Universal Robots URScript: Floor Straight.script

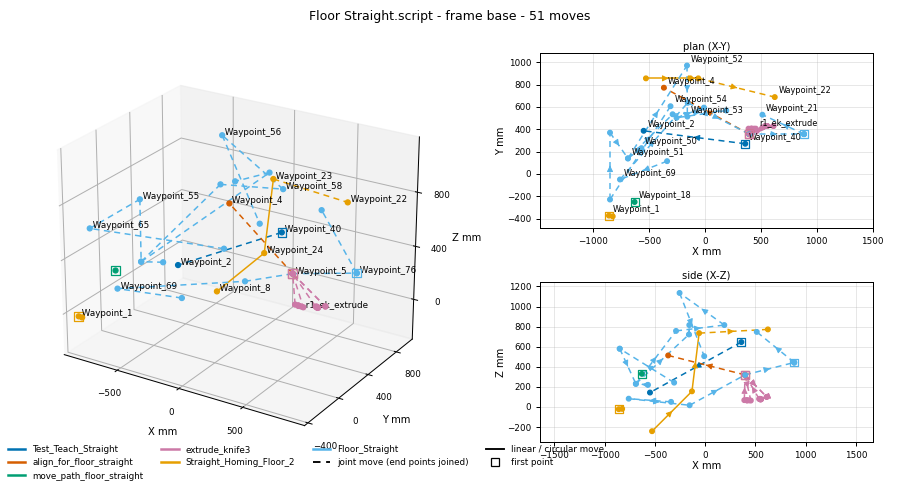
[picture p0: tool path of Floor Straight.script in frame base, 51 of 94 moves have a stored position in this frame; points joined in program order, loops and branches not executed]
def Floor_Straight():
  global _hidden_verificationVariable=0
  set_standard_analog_input_domain(0, 1)
  set_standard_analog_input_domain(1, 1)
  set_tool_analog_input_domain(0, 1)
  set_tool_analog_input_domain(1, 1)
  set_analog_outputdomain(0, 0)
  set_analog_outputdomain(1, 0)
  set_input_actions_to_default()
  set_target_payload(10.800000, [-0.001000, -0.053000, 0.068000], [0.081228, 0.081228, 0.081228, 0.000000, 0.000000, 0.000000])
  set_tool_communication(False, 115200, 0, 1, 1.5, 3.5)
  set_tool_output_mode(0)
  set_tool_digital_output_mode(0, 1)
  set_tool_digital_output_mode(1, 1)
  set_tool_voltage(0)
  set_tcp(p[-0.011699999999999999,-0.328,0.105,1.2092,-1.2092,1.2092])
  set_safety_mode_transition_hardness(1)
  set_gravity([0.0, 0.0, 9.82])
  global robot_number=3
  global Point_1=p[0.0,0.0,0.0,0.0,0.0,0.0]
  global Point_2=p[0.0,0.0,0.0,0.0,0.0,0.0]
  # begin: URCap Installation Node
  #   Source: UR Connect, 1.13.79, Universal Robots
  #   Type: UR Connect
  myurRPC = rpc_factory("xmlrpc","http://127.0.0.1:40474")
  # end: URCap Installation Node
  # begin: URCap Installation Node
  #   Source: MachineLogic for Universal Robots, 3.1.7, Vention Inc.
  #   Type: MachineLogic for Universal Robots
  def waitForResponse(expected_response_vention, cname_vention):
  response_vention = socket_read_string(cname_vention,timeout=15)
  while response_vention != expected_response_vention:
  sleep(0.01)
  response_vention = socket_read_string(cname_vention,timeout=15)
  end
  sleep(0.01)
  sync()
  end
  def sendString(string_vention, expected_response_vention, cname_vention):
  socket_send_string(str_cat(string_vention,";"), cname_vention)
  response_vention = socket_read_string(cname_vention,timeout=15)
  if(response_vention == "nAck"):
  popup("nAck received")
  end
  while response_vention != expected_response_vention:
  sleep(0.01)
  response_vention = socket_read_string(cname_vention,timeout=15)
  if(response_vention == "nAck"):
  popup("nAck received")
  end
  end
  sleep(0.01)
  sync()
  end
  def sendStringNAck(string_vention, expected_response_vention, cname_vention):
  socket_send_string(str_cat(string_vention,";"), cname_vention)
  response_vention = socket_read_string(cname_vention,timeout=15)
  if(response_vention == "nAck"):
  popup("nAck received")
  end
  while(response_vention != expected_response_vention and response_vention != "nAck"):
  sleep(0.01)
  response_vention = socket_read_string(cname_vention,timeout=15)
  if(response_vention == "nAck"):
  popup("nAck received",blocking=True)
  end
  end
  sleep(0.01)
  sync()
  end
  def sendStringWithTimeout(string_vention, expected_response_vention, cname_vention):
  socket_send_string(str_cat(string_vention,";"), cname_vention)
  response_vention = socket_read_string(cname_vention,timeout=10)
  if(response_vention == "nAck"):
  popup("nAck received"+string_vention)
  end
  sleep(0.01)
  sync()
  end
  def pollString(string_vention, expected_response_vention, cname_vention):
  socket_send_string(str_cat(string_vention,";"), cname_vention)
  response_vention = socket_read_string(cname_vention,timeout=15)
  if(response_vention == "nAck"):
  popup("nAck received")
  end
  while response_vention != expected_response_vention:
  sleep(1)
  socket_send_string(str_cat(string_vention,";"), cname_vention)
  response_vention = socket_read_string(cname_vention,timeout=15)
  if(response_vention == "nAck"):
  popup("nAck received")
  end
  end
  sleep(0.01)
  sync()
  end
  def sendVariable(var_vention, data_vention, expected_response_vention, cname_vention):
  socket_set_var(var_vention, data_vention, cname_vention)
  response_vention = socket_read_string(cname_vention,timeout=15)
  if(response_vention == "nAck"):
  popup("nAck received")
  end
  while response_vention != expected_response_vention:
  sleep(0.01)
  response_vention = socket_read_string(cname_vention,timeout=15)
  if(response_vention == "nAck"):
  popup("nAck received")
  end
  end
  sleep(0.01)
  sync()
  end
  def intToString(integer_vention,cname_vention):
  stringFix=""
  multiplier_vention123=1
  if integer_vention<0:
  stringFix="-"
  multiplier_vention123=-1
  end
  socket_set_var("GetString",integer_vention*multiplier_vention123,cname_vention)
  string_vention=""
  while string_vention=="":
  sleep(0.01)
  string_vention=socket_read_string(cname_vention,timeout=15)
  end
  sleep(0.01)
  sync()
  string_vention=stringFix+string_vention
  return string_vention
  end
  string_vention=""
  isVentionMovementBusy = False
  isVentionParallelMovementSendingScript = False
  ventionThreadHandle = 1
  isVentionMovementBusyMachineMotion1 = False
  isVentionParallelMovementSendingScriptMachineMotion1 = False
  socket_vention = socket_open("192.168.3.52", 9999, "MachineMotion1")
  if socket_vention==False:
  popup("Check configuration, can't connect to MachineMotion")
  end
  waitForResponse("MachineMotion connection established", "MachineMotion1")
  sendString("isReady", "MachineMotion isReady = true", "MachineMotion1")
  sendStringWithTimeout("setURCapVersion2", "setURCapVersion loaded", "MachineMotion1")
  sendString("SET speed_v2 1000000", "Ack", "MachineMotion1")
  sendString("SET acceleration_v2 100000", "Ack", "MachineMotion1")
  sendString("SET de_axis_1_microsteps_config 8", "Ack", "MachineMotion1")
  sendString("SET de_axis_1_mechanical_gain_config_v2 150000.0", "Ack", "MachineMotion1")
  sendString("SET de_axis_1_direction_config 1", "Ack", "MachineMotion1")
  sendString("SET de_axis_1_type_config Custom Actuator ", "Ack", "MachineMotion1")
  sendString("de_axis_1_config_exec", "Ack", "MachineMotion1")
  # end: URCap Installation Node
  # begin: URCap Installation Node
  #   Source: WireTank Serial, 4.9.0, WireTank, LLC
  #   Type: WireTank Serial
  WTSerialBridge = rpc_factory("xmlrpc","http://127.0.0.1:40511/RPC2")
  # end: URCap Installation Node
  step_count_93fcdbb1_1181_43ea_a7f0_580262fe9a13 = 0.0
  thread Step_Counter_Thread_773b6cc1_d8f8_46f9_9db1_b39c1ae6633a():
    while (True):
      step_count_93fcdbb1_1181_43ea_a7f0_580262fe9a13 = step_count_93fcdbb1_1181_43ea_a7f0_580262fe9a13 + 1.0
      sync()
    end
  end
  run Step_Counter_Thread_773b6cc1_d8f8_46f9_9db1_b39c1ae6633a()
  global free_dr_already=  False
  global freedrive_m_var=  False
  global Waypoint_76_p=p[.886939072471, .356263001241, .442999104957, 2.316306590719, 2.057646408592, .074101958719]
  global Waypoint_76_q=[-3.2647881984118814, -1.2522049299371645, 1.5824044773896437, 0.9175786249801816, -0.008369636028316307, -1.3112608249927966]
  global Waypoint_50_p=p[-.568711442653, .230601791901, .220208834751, -1.519093932087, -.535128035721, .573965472012]
  global Waypoint_50_q=[-0.021522347127095998, -1.2794721287539979, 2.4323821703540247, 5.090870934515753, -2.2996109167682093, 1.533644199371338]
  global Waypoint_51_p=p[-.689649894186, .139001107022, .230693120258, -.852023156701, -1.645963115617, 1.645984943001]
  global Waypoint_51_q=[-1.1454814116107386, -1.5427037247321387, 2.8454700152026575, 4.979047852545538, -4.902958456669943, 1.5718834400177002]
  global Waypoint_52_p=p[-.160992057407, .970528182050, .722037363514, -.554955923310, .106486629259, .328544950173]
  global Waypoint_52_q=[-1.2978580633746546, -1.3217003357461472, 2.2583277861224573, 3.7025129038044433, -2.952825371419088, 0.9627944231033325]
  global Waypoint_53_p=p[-.157624488365, .513351401913, .815670293526, -.672704566373, -1.852329693545, -.055423312366]
  global Waypoint_53_q=[-2.7676661650287073, -1.8206430874266566, 2.312763277684347, 1.0122546392628173, -1.0765226523028772, -0.8102834860431116]
  global Waypoint_54_p=p[-.308528116178, .606080777007, .242371251996, -2.133736658076, .349438277129, 2.130953356703]
  global Waypoint_54_q=[-1.9617512861834925, -1.2994225782207032, 2.207935158406393, 0.745708628291748, 1.5955500602722168, 1.41863214969635]
  global Waypoint_65_p=p[-.850299549699, -.229060500451, .580194265918, -.066683564301, -1.566406749139, -.045536147896]
  global Waypoint_65_q=[0.11527767777442932, -1.206728772526123, 2.660132948552267, 3.2525827127644042, -4.69939905801882, -0.18521625200380498]
  global Waypoint_55_p=p[-.850295942693, .369353811615, .580190947871, -.066690142153, -1.566409865149, -.045506050424]
  global Waypoint_55_q=[-0.89636737505068, -1.198587493305542, 2.6061368624316614, 3.3119169908710937, -4.700617257748739, 0.826545238494873]
  global Waypoint_59_p=p[-.689650832419, .138973473550, .230700469426, -.851985360280, -1.645991124348, 1.645990580233]
  global Waypoint_59_q=[-1.1454528013812464, -1.5427289356342335, 2.8454795519458216, 4.979044186859884, -4.902960960065023, 1.5718833208084106]
  global Waypoint_71_p=p[-.289684660393, .534258475721, .757199031184, -.295236718653, -.653013693815, .389426431276]
  global Waypoint_71_q=[-1.3941848913775843, -1.6550847492613734, 2.7336130777942103, 4.156678839320801, -3.798194471989767, 1.7310842275619507]
  global Waypoint_58_p=p[.191120239889, .567518478899, .815512910186, -.135765364935, .396070873472, .208834263225]
  global Waypoint_58_q=[-1.651280705128805, -1.7712346516051234, 2.617981735860006, 3.3066598612019042, -2.656208101903097, 0.8563313484191895]
  global Waypoint_56_p=p[-.254568281661, .502958752129, 1.135400507516, -.261908057482, -.749714619963, 1.349050618455]
  global Waypoint_56_q=[-2.0344861189471644, -1.9012485943236292, 2.469647232686178, 2.2012061315723876, -1.1677187124835413, -0.5094392935382288]
  global Waypoint_57_p=p[-.009221327687, .593713365169, .505808930157, -1.424394189587, -2.344106819810, -.527597949261]
  global Waypoint_57_q=[-2.920837704335348, -1.9932075939574183, 2.3856611887561243, 0.6815890508839111, -0.5688460508929651, -1.1506975332843226]
  global Waypoint_67_p=p[-.339169194335, .114271165560, .051007401747, -.434162127311, 1.872717119498, -1.885153895998]
  global Waypoint_67_q=[-1.410516087208883, -0.9778240484050293, 2.47756010690798, -1.72361483196401, -0.3956816832171839, 1.808600902557373]
  global Waypoint_69_p=p[-.760826542313, -.049762698068, .082649581767, -1.026233921905, -1.612699318499, 1.547123897415]
  global Waypoint_69_q=[-0.22154647508730108, -1.118469015961029, 2.7561236063586634, -1.5568565337783475, -3.851987902318136, 1.559481143951416]
  global Waypoint_70_p=p[-.154414768496, .636923137577, .016979120256, -.302753655748, 1.486961848367, .122240024639]
  global Waypoint_70_q=[-1.1281922499286097, -1.0678585332683106, 2.4290812651263636, -2.7994214497008265, -1.6034835020648401, 1.7401196956634521]
  global Waypoint_49_p=p[.397354147848, .356263001249, .319808682466, 2.316306590727, 2.057646408591, .074101958728]
  global Waypoint_49_q=[-3.4579480330096644, -2.0568953953185023, 2.3266006151782435, -0.2270372670939942, -0.1993797461139124, -0.10534602800478154]
  global Waypoint_75_p=p[.886939072471, .356263001241, .442999104957, 2.316306590719, 2.057646408592, .074101958719]
  global Waypoint_75_q=[-3.2647881984118814, -1.2522049299371645, 1.5824044773896437, 0.9175786249801816, -0.008369636028316307, -1.3112608249927966]
  global Waypoint_21_p=p[.514110621997, .530257197556, .747563358129, .126585912537, 2.198134649130, 2.122774364636]
  global Waypoint_21_q=[-3.3739228671287087, -1.9731126642389452, 2.1046588209607195, -0.4109766241583843, -0.11921991224173922, 0.2750749283180509]
  global Waypoint_40_p=p[.360688403366, .270119715397, .646144746546, .057805349154, 2.125995180379, 2.134053153683]
  global Waypoint_40_q=[-3.4579489866839808, -2.0569035015501917, 2.3265796343432825, -0.22706706941638188, -0.1993501822101038, -0.10534793535341436]
  global Waypoint_2_p=p[-.548957282596, .386284559177, .143710178207, 1.570800598292, -.000025190822, .000004803470]
  global Waypoint_2_q=[-1.0516188780414026, -1.010990933781006, 2.1562450567828577, -1.143702046280243, -1.0526168982135218, -0.0017235914813440445]
  global Waypoint_5_p=p[.397354147848, .356263001249, .319808682466, 2.316306590727, 2.057646408591, .074101958728]
  global Waypoint_5_q=[-3.461131359466087, -2.062322244150579, 2.329180664349958, -0.21922739695102145, -0.20100694585188528, -0.11040669743860754]
  global Waypoint_4_p=p[-.367892231714, .771855800230, .513016861312, -2.038498198230, .435742020455, 2.027527731542]
  global Waypoint_4_q=[-1.785487476979391, -1.7826982937254847, 2.1989410559283655, -1.9407421551146449, -1.5771468321429651, -1.4076789061175745]
  global Waypoint_18_p=p[-.629785486869, -.251121069656, .329949691670, 2.361287469623, -.065058504799, -1.958677600219]
  global Waypoint_18_q=[0.031418071511559086, -2.137055665484551, 2.546713757031022, -1.7951564170717766, -1.4854111175142606, 0.0015551912058106448]
  global r1_ek_oldhome_p=p[.397380247322, .356253634699, .319820846021, 2.316316320871, 2.057594704604, .074118471609]
  global r1_ek_oldhome_q=[-3.457949940358297, -2.056894441644186, 2.32658034959902, -0.2270551484874268, -0.19935208955873662, -0.10533696809877569]
  global r1_ek_extrude_p=p[.454852104155, .405448828659, .064015413765, 2.316807606413, 2.051392071696, .076664825947]
  global r1_ek_extrude_q=[-3.274653975163595, -1.5604325172356148, 2.467809502278463, -0.34438879907641606, -0.014281574879781544, -0.6303489843951624]
  global r1_ek_front_p=p[.439064809878, .405452261046, .065996139932, 2.316843937268, 2.051427632497, .076607106393]
  global r1_ek_front_q=[-3.280560557042257, -1.6287623844542445, 2.502561871205465, -0.47416289270434575, -0.019731823598043263, -0.4669149557696741]
  global r1_ek_middle_p=p[.419010105608, .404850828431, .065994665459, 2.309574128677, 2.044678176343, .089098333896]
  global r1_ek_middle_q=[-3.290863100682394, -1.70143522838735, 2.548208538685934, -0.589385525589325, -0.029501263295308888, -0.3372734228717249]
  global r1_ek_middle2_p=p[.417011768852, .405435328663, .065002627117, 2.316867113472, 2.051334925313, .076628493429]
  global r1_ek_middle2_q=[-3.289830032979147, -1.6934038601317347, 2.5445857683764856, -0.579618052845337, -0.028589550648824513, -0.33885270753969365]
  global r1_ek_bottom_p=p[.413071667620, .405431286494, .067999701073, 2.316819721954, 2.051304037200, .076688572349]
  global r1_ek_bottom_q=[-3.2916205565081995, -1.708447118798727, 2.5485368410693567, -0.5849895042232056, -0.03033763567079717, -0.32244998613466436]
  global r1_ek_end_p=p[.389998638281, .405443674081, .068004818811, 2.316851991921, 2.051367741778, .076612018685]
  global r1_ek_end_q=[-3.3030064741717737, -1.7640062771239222, 2.5831297079669397, -0.63420523822818, -0.04154044786562139, -0.2521465460406702]
  global r2_ek_oldhome_p=p[.397380247322, .356253634699, .319820846021, 2.316316320871, 2.057594704604, .074118471609]
  global r2_ek_oldhome_q=[-3.461132842686933, -2.062320779349874, 2.32916033290004, -0.21924456446492258, -0.20097883707844666, -0.11039879152527199]
  global r2_ek_extrude_p=p[.612885745678, .429305279732, .100477107124, 2.149994969793, 2.225764025207, .087353352584]
  global r2_ek_extrude_q=[-3.199475796455825, -1.4862854517875999, 2.263543898005424, -0.6928175084157413, -0.09183293866530295, -0.15653548683830643]
  global r2_ek_front_p=p[.556405415915, .429305279815, .076984362723, -2.170411249256, -2.268200695165, -.015853660170]
  global r2_ek_front_q=[-3.2029012478485694, -1.4943971905029905, 2.3176866046272355, -0.727203417516419, -0.10461513056100813, -0.1013922369747533]
  global r2_ek_middle_p=p[.550033970532, .429305279917, .076253920653, -2.170411249261, -2.268200695170, -.015853660159]
  global r2_ek_middle_q=[-3.2036200175167613, -1.5006788185274456, 2.326226188945654, -0.730095076239345, -0.10533288811000929, -0.10075548926859312]
  global r2_ek_bottom_p=p[.546594660555, .429305280025, .080868477599, -2.170411249265, -2.268200695174, -.015853660149]
  global r2_ek_bottom_q=[-3.204010221105431, -1.5099366263094405, 2.3272215014458872, -0.722096275899732, -0.10572512264357048, -0.10049057923478166]
  global r2_ek_end_p=p[.537335106646, .429305280055, .080868477459, -2.170411249266, -2.268200695175, -.015853660146]
  global r2_ek_end_q=[-3.205098875769389, -1.5204959829395506, 2.3387656715508855, -0.724001524008818, -0.10681294496314919, -0.09956563917089412]
  def calculate_point_to_move_towards(feature, direction, position_distance):
    local posDir=[direction[0], direction[1], direction[2]]
    if (norm(posDir) < 1e-6):
      return get_target_waypoint()
    end
    local direction_vector_normalized=normalize(posDir)
    local displacement_pose=p[direction_vector_normalized[0] * position_distance,direction_vector_normalized[1] * position_distance,direction_vector_normalized[2] * position_distance,0,0,0]
    local wanted_displacement_in_base_frame=pose_sub(pose_trans(feature, displacement_pose), feature)
    return pose_add(get_target_waypoint(), wanted_displacement_in_base_frame)
  end
  global Waypoint_1_p=p[-.859669104529, -.373308604741, -.021871009822, 1.209000000000, -1.209000000000, -1.209000000000]
  global Waypoint_1_q=[0.3601058940048852, -0.8464386020098615, 2.4787281289145255, -1.6334201935107835, 1.9316825434161362, -3.384850340317769E-4]
  global Waypoint_6_p=p[-.826115368487, -.379847833008, -.018789706596, -.053757400051, -.080726049716, 1.170328425587]
  global Waypoint_6_q=[0.20623618383850975, -0.037244073839099556, 1.8264915282007301, -3.2712711586447565, 1.5882864721468046, 2.5367371432461816]
  global Waypoint_8_p=p[-.528586726350, .855731167328, -.241098719203, -.034347324650, -.041760335369, -1.096045309072]
  global Waypoint_8_q=[-1.2365026682154365, 0.21046607420950655, 1.414738542801075, -3.145403886739818, 1.5693855394695468, 1.7112884178826036]
  global Waypoint_24_p=p[-.131140323045, .855731167178, .156011078035, -.034347324657, -.041760335378, -1.096045309072]
  global Waypoint_24_q=[-1.6817946855399448, -0.23042096439631443, 2.0400888245341187, -3.3348765239674023, 1.5472825176858356, 2.15593654853991]
  global Waypoint_23_p=p[-.059797728511, .855731167376, .735189988230, -.034347324653, -.041760335373, -1.096045309072]
  global Waypoint_23_q=[-1.7671370912445887, -1.0666469027155046, 2.2956126081674424, -2.756218919979178, 1.544098900974971, 2.2408582527447005]
  global Waypoint_22_p=p[.624813144152, .687861929675, .772422833303, .126119483886, 2.325670393286, 2.041529927887]
  global Waypoint_22_q=[-3.0457660852497743, -1.59044931348798, 1.7566404370712891, 0.44788167229645204, 0.2257630446261064, -0.5814331872529142]
  def Test_Teach_Straight():
    $ 136 "Test_Teach_Straight" "noBreak"
    $ 137 "Set"
    set_tcp(p[1.4000000000000001E-4,-0.01751,0.285,0.0,0.0,0.0])
    $ 141 "MoveJ"
    $ 142 "Waypoint_40" "breakAfter"
    set_tcp(p[0.0,0.0,0.019,0.0,0.0,0.0])
    movej(get_inverse_kin(Waypoint_40_p, qnear=Waypoint_40_q), a=1.3962634015954636, v=1.0471975511965976)
    $ 143 "'above waypoint is home'"
    # 'above waypoint is home'
    $ 144 "Waypoint_2" "breakAfter"
    set_tcp(p[0.0,0.0,0.019,0.0,0.0,0.0])
    movej(get_inverse_kin(Waypoint_2_p, qnear=Waypoint_2_q), a=1.3962634015954636, v=1.0471975511965976)
    $ 145 "Set"
    set_tcp(p[1.4000000000000001E-4,-0.01751,0.285,0.0,0.0,0.0])
    $ 146 "freedrive_m_var≔ False "
    global freedrive_m_var=  False
    $ 147 "freedrive_m_var≔ True "
    global freedrive_m_var=  True
    $ 148 "Popup: Move the TCP to the left side of the weld (very end of the V chisel), then click 'Continue'"
    popup("Move the TCP to the left side of the weld (very end of the V chisel), then click 'Continue'", "Message", False, False, blocking=True)
    $ 149 "tcp_pose_left≔get_actual_tcp_pose()"
    global tcp_pose_left= get_actual_tcp_pose ()
    $ 150 "Popup: Move the TCP to the right side of the weld (very end of the V chisel), then click 'Continue'"
    popup("Move the TCP to the right side of the weld (very end of the V chisel), then click 'Continue'", "Message", False, False, blocking=True)
    $ 151 "tcp_pose_right≔get_actual_tcp_pose()"
    global tcp_pose_right= get_actual_tcp_pose ()
    $ 152 "freedrive_m_var≔ False "
    global freedrive_m_var=  False
    $ 153 "Wait: 0.25"
    sleep(0.25)
    $ 154 "sync()"
    sync()
  end
  def align_for_floor_straight():
    $ 155 "align_for_floor_straight" "noBreak"
    $ 161 "MoveJ"
    $ 162 "Waypoint_5" "breakAfter"
    movej(get_inverse_kin(Waypoint_5_p, qnear=Waypoint_5_q), a=1.3962634015954636, v=1.0471975511965976)
    $ 164 "Waypoint_4" "breakAfter"
    movej(get_inverse_kin(Waypoint_4_p, qnear=Waypoint_4_q), a=1.3962634015954636, v=1.0471975511965976)
  end
  def move_path_floor_straight():
    $ 169 "move_path_floor_straight" "noBreak"
    $ 170 "p1≔pathturn[1]"
    global p1=pathturn[1]
    $ 171 "p2≔pathturn[2]"
    global p2=pathturn[2]
    $ 172 "p3≔pathturn[3]"
    global p3=pathturn[3]
    $ 173 "p4≔pathturn[4]"
    global p4=pathturn[4]
    $ 174 "p5≔pathturn[5]"
    global p5=pathturn[5]
    $ 175 "p6≔pathturn[6]"
    global p6=pathturn[6]
    $ 176 "pa1≔p[p1[0]+0.05,p1[1],p1[2],p1[3],p1[4],p1[5]]"
    global pa1=p[p1[0]+0.05,p1[1],p1[2],p1[3],p1[4],p1[5]]
    $ 177 "pret≔p[p6[0]+0.05,p6[1],p6[2],p6[3],p6[4],p6[5]]"
    global pret=p[p6[0]+0.05,p6[1],p6[2],p6[3],p6[4],p6[5]]
    $ 178 "pret2≔p[-0.81,p6[1],p6[2],p6[3],p6[4],p6[5]]"
    global pret2=p[-0.81,p6[1],p6[2],p6[3],p6[4],p6[5]]
    $ 179 "'go to preheat'"
    # 'go to preheat'
    $ 180 "Set"
    set_tcp(p[-0.011699999999999999,-0.328,0.105,1.2092,-1.2092,1.2092])
    $ 181 "MoveJ"
    $ 182 "pa1" "breakAfter"
    movej(pa1, a=1.3962634015954636, v=1.0471975511965976)
    $ 183 "MoveL"
    $ 184 "p1" "breakAfter"
    movel(p1, a=0.05, v=0.05)
    $ 185 "Wait: 4.0"
    sleep(4.0)
    # begin: URCap Program Node
    #   Source: WireTank Serial, 4.9.0, WireTank, LLC
    #   Type: WireTank Serial
    $ 186 "Serial Bridge uR1"
    SerialResponse = WTSerialBridge.send_command("/dev/ttyUSB0",1200, 8, "None", "One", "None", 1000, "None", "None", [252,82,49], False)
    # end: URCap Program Node
    $ 187 "Set DO[0]=On"
    set_standard_digital_out(0, True)
    $ 188 "Wait: 1.0"
    sleep(1.0)
    $ 189 "MoveL"
    $ 190 "p2" "breakAfter"
    movel(p2, a=1.2, v=0.01)
    $ 191 "p3" "breakAfter"
    movel(p3, a=1.2, v=0.01)
    $ 192 "p4" "breakAfter"
    movel(p4, a=1.2, v=0.01)
    $ 193 "p5" "breakAfter"
    movel(p5, a=1.2, v=0.01)
    # begin: URCap Program Node
    #   Source: WireTank Serial, 4.9.0, WireTank, LLC
    #   Type: WireTank Serial
    $ 194 "Serial Bridge uR0"
    SerialResponse = WTSerialBridge.send_command("/dev/ttyUSB0",1200, 8, "None", "One", "None", 1000, "None", "None", [252,82,48], False)
    # end: URCap Program Node
    $ 195 "Set DO[0]=Off"
    set_standard_digital_out(0, False)
    $ 196 "MoveL"
    $ 197 "p6" "breakAfter"
    movel(p6, a=1.2, v=0.01)
    $ 198 "Wait: 1.0"
    sleep(1.0)
    $ 199 "MoveL"
    $ 200 "pret" "breakAfter"
    movel(pret, a=0.05, v=0.05)
    $ 201 "pret2" "breakAfter"
    movel(pret2, a=0.05, v=0.05)
    $ 202 "MoveJ"
    $ 203 "Waypoint_18" "breakAfter"
    movej(get_inverse_kin(Waypoint_18_p, qnear=Waypoint_18_q), a=1.3962634015954636, v=1.0471975511965976)
  end
  def extrude_knife3():
    $ 204 "extrude_knife3" "noBreak"
    $ 205 "pre program stuff"
    $ 206 "Set"
    set_tcp(p[-0.011699999999999999,-0.328,0.105,1.2092,-1.2092,1.2092])
    $ 207 "ek_sp≔get_actual_tcp_pose()"
    global ek_sp= get_actual_tcp_pose ()
    $ 208 "MoveL"
    $ 209 "ek_sp" "breakAfter"
    movel(ek_sp, a=1.2, v=0.005)
    $ 211 "'list possible points'"
    # 'list possible points'
    $ 212 "robot 1 moves"
    $ 213 "If 1≟2"
    if (1 == 2):
      $ 214 "MoveJ"
      $ 215 "r1_ek_oldhome" "breakAfter"
      movej(get_inverse_kin(r1_ek_oldhome_p, qnear=r1_ek_oldhome_q), a=1.3962634015954636, v=1.0471975511965976)
      $ 216 "r1_ek_extrude" "breakAfter"
      movej(get_inverse_kin(r1_ek_extrude_p, qnear=r1_ek_extrude_q), a=1.3962634015954636, v=1.0471975511965976)
      $ 217 "r1_ek_front" "breakAfter"
      movej(get_inverse_kin(r1_ek_front_p, qnear=r1_ek_front_q), a=1.3962634015954636, v=1.0471975511965976)
      $ 218 "r1_ek_middle" "breakAfter"
      movej(get_inverse_kin(r1_ek_middle_p, qnear=r1_ek_middle_q), a=1.3962634015954636, v=1.0471975511965976)
      $ 219 "r1_ek_middle2" "breakAfter"
      movej(get_inverse_kin(r1_ek_middle2_p, qnear=r1_ek_middle2_q), a=1.3962634015954636, v=1.0471975511965976)
      $ 220 "r1_ek_bottom" "breakAfter"
      movej(get_inverse_kin(r1_ek_bottom_p, qnear=r1_ek_bottom_q), a=1.3962634015954636, v=1.0471975511965976)
      $ 221 "r1_ek_end" "breakAfter"
      movej(get_inverse_kin(r1_ek_end_p, qnear=r1_ek_end_q), a=1.3962634015954636, v=1.0471975511965976)
    end
    $ 222 "robot 2 moves"
    $ 223 "If 1≟2"
    if (1 == 2):
      $ 224 "MoveJ"
      $ 225 "r2_ek_oldhome" "breakAfter"
      movej(get_inverse_kin(r2_ek_oldhome_p, qnear=r2_ek_oldhome_q), a=1.3962634015954636, v=1.0471975511965976)
      $ 227 "r2_ek_extrude" "breakAfter"
      movej(get_inverse_kin(r2_ek_extrude_p, qnear=r2_ek_extrude_q), a=1.3962634015954636, v=1.0471975511965976)
      $ 228 "r2_ek_front" "breakAfter"
      movej(get_inverse_kin(r2_ek_front_p, qnear=r2_ek_front_q), a=1.3962634015954636, v=1.0471975511965976)
      $ 229 "r2_ek_middle" "breakAfter"
      movej(get_inverse_kin(r2_ek_middle_p, qnear=r2_ek_middle_q), a=1.3962634015954636, v=1.0471975511965976)
      $ 230 "r2_ek_bottom" "breakAfter"
      movej(get_inverse_kin(r2_ek_bottom_p, qnear=r2_ek_bottom_q), a=1.3962634015954636, v=1.0471975511965976)
      $ 231 "r2_ek_end" "breakAfter"
      movej(get_inverse_kin(r2_ek_end_p, qnear=r2_ek_end_q), a=1.3962634015954636, v=1.0471975511965976)
    end
    $ 232 "'detemine correct points for which robot'"
    # 'detemine correct points for which robot'
    $ 233 "If robot_number≟1"
    if (robot_number == 1):
      $ 234 "robot1 positions"
      $ 235 "ek_oldhome≔r1_ek_oldhome_p"
      global ek_oldhome=r1_ek_oldhome_p
      $ 236 "ek_extrude≔r1_ek_extrude_p"
      global ek_extrude=r1_ek_extrude_p
      $ 237 "ek_front≔r1_ek_front_p"
      global ek_front=r1_ek_front_p
      $ 238 "ek_middle≔r1_ek_middle_p"
      global ek_middle=r1_ek_middle_p
      $ 239 "ek_middle2≔r1_ek_middle2_p"
      global ek_middle2=r1_ek_middle2_p
      $ 240 "ek_bottom≔r1_ek_bottom_p"
      global ek_bottom=r1_ek_bottom_p
      $ 241 "ek_end≔r1_ek_end_q"
      global ek_end=r1_ek_end_q
    else:
      $ 242 "ElseIf robot_number≟2"
      if (robot_number == 2):
        $ 243 "robot1 positions"
        $ 244 "ek_oldhome≔r2_ek_oldhome_p"
        global ek_oldhome=r2_ek_oldhome_p
        $ 245 "ek_extrude≔r2_ek_extrude_p"
        global ek_extrude=r2_ek_extrude_p
        $ 246 "ek_front≔r2_ek_front_p"
        global ek_front=r2_ek_front_p
        $ 247 "ek_middle≔r2_ek_middle_p"
        global ek_middle=r2_ek_middle_p
        $ 248 "ek_middle2≔r2_ek_middle_p"
        global ek_middle2=r2_ek_middle_p
        $ 249 "ek_bottom≔r2_ek_bottom_p"
        global ek_bottom=r2_ek_bottom_p
        $ 250 "ek_end≔r2_ek_end_q"
        global ek_end=r2_ek_end_q
      end
    end
    $ 251 "'start of program'"
    # 'start of program'
    $ 253 "Set"
    set_tcp(p[-0.011699999999999999,-0.328,0.105,1.2092,-1.2092,1.2092])
    $ 254 "MoveJ"
    $ 256 "ek_oldhome" "breakAfter"
    movej(ek_oldhome, a=1.3962634015954636, v=1.0471975511965976)
    $ 257 "'above waypoint is home'"
    # 'above waypoint is home'
    $ 258 "'move above bucket'"
    # 'move above bucket'
    $ 259 "MoveJ"
    $ 261 "ek_extrude" "breakAfter"
    movej(ek_extrude, a=1.3962634015954636, v=1.0471975511965976)
    $ 262 "'extrude out a foot'"
    # 'extrude out a foot'
    # begin: URCap Program Node
    #   Source: WireTank Serial, 4.9.0, WireTank, LLC
    #   Type: WireTank Serial
    $ 264 "Serial Bridge uR1"
    SerialResponse = WTSerialBridge.send_command("/dev/ttyUSB0",1200, 8, "None", "One", "None", 1000, "None", "None", [252,82,49], False)
    # end: URCap Program Node
    $ 265 "Set DO[0]=On"
    set_standard_digital_out(0, True)
    $ 266 "Wait: 24.0"
    sleep(24.0)
    # begin: URCap Program Node
    #   Source: WireTank Serial, 4.9.0, WireTank, LLC
    #   Type: WireTank Serial
    $ 267 "Serial Bridge uR0"
    SerialResponse = WTSerialBridge.send_command("/dev/ttyUSB0",1200, 8, "None", "One", "None", 1000, "None", "None", [252,82,48], False)
    # end: URCap Program Node
    $ 268 "Wait: 1.0"
    sleep(1.0)
    $ 269 "Set DO[0]=Off"
    set_standard_digital_out(0, False)
    $ 270 "'slice'"
    # 'slice'
    $ 271 "MoveL"
    $ 277 "ek_front" "breakAfter"
    movel(ek_front, a=0.05, v=0.03)
    $ 278 "ek_middle" "breakAfter"
    movel(ek_middle, a=0.05, v=0.03)
    $ 279 "ek_middle2" "breakAfter"
    movel(ek_middle2, a=0.05, v=0.03)
    $ 280 "ek_bottom" "breakAfter"
    movel(ek_bottom, a=0.05, v=0.03)
    $ 281 "ek_end" "breakAfter"
    movel(ek_end, a=0.05, v=0.03)
    $ 282 "MoveJ"
    $ 284 "ek_oldhome" "breakAfter"
    movej(ek_oldhome, a=1.3962634015954636, v=1.0471975511965976)
    $ 285 "'above waypoint is home'"
    # 'above waypoint is home'
  end
  def Straight_Homing_Floor_2():
    $ 287 "Straight_Homing_Floor_2" "noBreak"
    $ 288 "Set"
    set_tcp(p[1.4000000000000001E-4,-0.01751,0.285,0.0,0.0,0.0])
    $ 289 "'dummy move below for debug'"
    # 'dummy move below for debug'
    $ 302 "Wait: 1.0"
    sleep(1.0)
    $ 304 "Script: analyze_touchpoints.script"
    # this file creates the function for analyzing touchpoints
    # define pi
    pi = 3.1415926535
    # initialize a lift column extension needed of 0.0
    global liftcolumnzneeded = 0.0 # set this variable in mm

    # this is the main entry point for calculations.
    # it takes in the 5 points, analyzes the shape of the box, and then calculates path points and returns them
    # specifically for Down, Over, then Around (DOtA)
    # specifically for right-sided boxes (vertical weld on right side of edge)
    def main_calculate_right(p11, p12, p21, p22, p3, p13, p23, chamferover):
        struct1 = analyze_touchpoints_only(p11, p12, p21, p22, p3)
        list1 = analyze_vertical_touchpoints(p11, p12, p13, p21, p22, p23, p3)
        struct2 = calculate_DOtA_points_right(struct1, list1, chamferover)
        validity = check_validity_right(struct1, struct2)
        return struct2
    end

    # this is the main entry point for calculations.
    # it takes in the 5 points, analyzes the shape of the box, and then calculates path points and returns them
    # specifically for Down, Over, then Around (DOtA)
    # specifically for left-sided boxes (vertical weld on left side of edge)
    def main_calculate_left(p11, p12, p21, p22, p3, p13, p23, chamferover):
        struct1 = analyze_touchpoints_only(p11, p12, p21, p22, p3)
        list1 = analyze_vertical_touchpoints(p11, p12, p13, p21, p22, p23, p3)
        struct2 = calculate_DOtA_points_left(struct1, list1, chamferover)
        validity = check_validity_left(struct1, struct2)
        return struct2
    end

    # this is the main entry point for calculations, for Floor Corner Extended.
    # it takes in the 7 touchpoints, analyzes the shape of the box.
    # takes in the user defined point for the top of the weld (tcp_pose_top) and then calculates path points
    # loopingly tries to calculate the extension along the sidewall that fulfills get_inverse_kin_has_solution() and provides the farthest extension possible
    # returns the pathpoints
    # specifically for Down, Over, then Around (DOtA)
    # specifically for right-sided boxes (vertical weld on right side of edge)
    def main_calculate_right_extended(p11, p12, p21, p22, p3, p13, p23, chamferover, chamferup, tcp_pose_top):
        struct1 = analyze_touchpoints_only(p11, p12, p21, p22, p3)
        list1 = analyze_vertical_touchpoints(p11, p12, p13, p21, p22, p23, p3)
        struct2 = calculate_DOtA_points_right_extended(struct1, list1, chamferover, chamferup, tcp_pose_top)
        struct3 = check_validity_right(struct1, struct2)
        return struct3
    end

    # this is the main entry point for calculations, for Floor Corner Extended.
    # it takes in the 7 touchpoints, analyzes the shape of the box.
    # takes in the user defined point for the top of the weld (tcp_pose_top) and then calculates path points
    # loopingly tries to calculate the extension along the sidewall that fulfills get_inverse_kin_has_solution() and provides the farthest extension possible
    # returns the pathpoints
    # specifically for Down, Over, then Around (DOtA)
    # specifically for left-sided boxes (vertical weld on left side of edge)
    def main_calculate_left_extended(p11, p12, p21, p22, p3, p13, p23, chamferover, chamferup, tcp_pose_top):
        struct1 = analyze_touchpoints_only(p11, p12, p21, p22, p3)
        list1 = analyze_vertical_touchpoints(p11, p12, p13, p21, p22, p23, p3)
        struct2 = calculate_DOtA_points_left_extended(struct1, list1, chamferover, chamferup, tcp_pose_top)
        struct3 = check_validity_left(struct1, struct2)
        return struct3
    end

    # it takes 5 arguments as points
    # it returns a struct containing: (pointintersect, pointapproach1, pointapproach2, point1, point2, point3, point4, point5, pointreturn1, heading1, heading2, heading3, path2r1, path2r2, path2l1, path2l2)
    # specifically for Around then Up (AtU)
    def analyze_touchpoints(p11, p12, p21, p22, p3):
      # FIND THE INTERSECTION
      # comment get the z
      zcoord=p3[2]

      # get the raw points from the first line
      l1p1x=p11[0]
      l1p1y=p11[1]
      l1p2x=p12[0]
      l1p2y=p12[1]

      # equate the first line in 2d space
      ml1 = (l1p2y-l1p1y) / (l1p2x-l1p1x)

      # b = y - mx
      bl1 = l1p1y - ml1 * l1p1x

      # get the raw points from the second line
      l2p1x=p21[0]
      l2p1y=p21[1]
      l2p2x=p22[0]
      l2p2y=p22[1]

      # equate the second line in 2d space
      ml2 = (l2p2y-l2p1y) / (l2p2x-l2p1x)

      # b = y - mx
      bl2 = l2p1y - ml2 * l2p1x


      # find the intersection of the two lines
      # m1x+b1 = m2x+b2
      # m1x - m2x = b2 - b1
      # x = (b2-b1) / (m1-m2)
      xintersect = (bl2-bl1) / (ml1-ml2)
      yintersect = ml1 * xintersect + bl1

      #FIND THE VECTORS
      #define a vector from the intersection to the second point on the first line
      l1delxfull = l1p2x - xintersect
      l1delyfull = l1p2y - yintersect

      l1delmag = sqrt(l1delxfull*l1delxfull + l1delyfull*l1delyfull)

      l1delxunit = l1delxfull / l1delmag
      l1delyunit = l1delyfull / l1delmag

      #define a vector from the intersection to the second point on the second line
      l2delxfull = l2p2x - xintersect
      l2delyfull = l2p2y - yintersect

      l2delmag = sqrt(l2delxfull*l2delxfull + l2delyfull*l2delyfull)

      l2delxunit = l2delxfull / l2delmag
      l2delyunit = l2delyfull / l2delmag

      # FIND THE FOUR POINTS ON THE LINES
      # find locations 8 inches away from  intersect point
      # CONST
      welddistance = 8
      roundoverdistance = 0.05
      zup = .375
      # inches
      wd = welddistance * 25.4 / 1000
      rod = roundoverdistance * 25.4 / 1000
      zup = zup * 25.4 / 1000

      # now we have the unit vector. extend the weld distance from the intersection
      x = xintersect + l1delxunit * wd
      y = yintersect + l1delyunit * wd
      z = zcoord + zup

      point1 = p[x,y,z,1.570796,0,0] # dummy orientation for now

      x = xintersect + l1delxunit * rod
      y = yintersect + l1delyunit * rod

      point2 = p[x,y,z,1.570796,0,0]

      # now we have the unit vector. extend the weld distance from the intersection
      x = xintersect + l2delxunit * wd
      y = yintersect + l2delyunit * wd

      point5 = p[x,y,z,0,-1.570796,0]

      x = xintersect + l2delxunit * rod
      y = yintersect + l2delyunit * rod

      point4 = p[x,y,z,0,-1.570796,0]

      #DEFINE APPROACH POINTS
      pointintersect = p[xintersect,yintersect,zcoord,0,0,0]
      pointapproach1 = p[xintersect+0.1,yintersect+0.1,z,1.570796,0,0]
      pointapproach2 = p[point1[0], point1[1]+0.1, point1[2], point1[3], point1[4], point1[5]]
      pointreturn1 = p[point5[0]+0.1, point5[1], point5[2], point5[3], point5[4], point5[5]]

      #FIND HEADINGS
      #for each heading, find the angle of the line with respect to the pos x axis. then add/subtract 90 degrees because you want to be perpendicular to that
      headingvector1 = convert_uv_to_heading(l1delxunit, l1delyunit)
      headingvector2 = convert_uv_to_heading(l2delxunit, l2delyunit)
      # find halfway heading
      heading2 = (headingvector1 + headingvector2)/2
      # find headings that the robot should face while traveling, perpendicular to the vectors of the sides of the box
      heading1 = headingvector1 + pi/2
      heading3 = headingvector2 - pi/2

      #FIND POINT 3
      #see if we have to / can find point 3
      findpoint3 = True
      if roundoverdistance == 0:
        findpoint3 = False
      end
      if findpoint3:
        # i need to find the point3 such that the arc from p2 to p3 to p4 is tangent to p1-p2 and p4-p5. making this a smooth path will be good
        # the direction of movement is from pointintersect in the direction of heading2
        # how much movement though? this will depend on whether it is actually a 90 degree angle or not.
        # first, find the perpendicular lines through points 2 and 4
        perp2 = find_perpendicular_line(ml1, point2[0], point2[1])
        perp4 = find_perpendicular_line(ml2, point4[0], point4[1])
        # next, find the intersection of those two lines
        perpintersect = find_intersection(perp2[0], perp2[1], perp4[0], perp4[1])
        radiusofcircle = distance_between(perpintersect[0], perpintersect[1], 0, point2[0], point2[1], 0)
        # find a vector the direction of heading2
        uvx = cos(heading2)
        uvy = sin(heading2)
        # compute point3. pass in negative radius because the direction is into the tank but we want to move from the intersection out to the rounded edge
        point3coords = add_vectordistance_to_point(perpintersect[0], perpintersect[1], z, uvx, uvy, 0, -1 * radiusofcircle)
        point3 = p[point3coords[0], point3coords[1], point3coords[2], 0, 0, 0]
      end

      #APPLY ACTUAL RXRYRZ TO POINTS
      # convert the headings to rxryrz and insert those values into the relevant points
      rxryrz = convert_heading_to_axang(heading1)
      rx = rxryrz[0]
      ry = rxryrz[1]
      rz = rxryrz[2]
      pointapproach1 = p[pointapproach1[0], pointapproach1[1], pointapproach1[2], rx, ry, rz]
      pointapproach2 = p[pointapproach2[0], pointapproach2[1], pointapproach2[2], rx, ry, rz]
      point1 = p[point1[0], point1[1], point1[2], rx, ry, rz]
      point2 = p[point2[0], point2[1], point2[2], rx, ry, rz]
      rxryrz = convert_heading_to_axang(heading2)
      rx = rxryrz[0]
      ry = rxryrz[1]
      rz = rxryrz[2]
      if findpoint3:
        point3 = p[point3[0], point3[1], point3[2], rx, ry, rz]
      else:
        point3 = point2
      end
      rxryrz = convert_heading_to_axang(heading3)
      rx = rxryrz[0]
      ry = rxryrz[1]
      rz = rxryrz[2]
      point4 = p[point4[0], point4[1], point4[2], rx, ry, rz]
      point5 = p[point5[0], point5[1], point5[2], rx, ry, rz]
      pointreturn1 = p[pointreturn1[0], pointreturn1[1], pointreturn1[2], rx, ry, rz]

      #find path2 (the part that goes up)
      four_vertical_points = find_vertical_points(pointintersect, l1delxunit, l1delyunit, l2delxunit, l2delyunit, zup, wd, heading1, heading3)
      path2r1 = four_vertical_points[0]
      path2r2 = four_vertical_points[1]
      path2l1 = four_vertical_points[2]
      path2l2 = four_vertical_points[3]

      #RETURN STRUCT
      ret = struct(pointintersect=pointintersect, pointapproach1=pointapproach1, pointapproach2=pointapproach2, point1=point1, point2=point2, point3=point3, point4=point4, point5=point5, pointreturn1=pointreturn1, heading1=heading1, heading2=heading2, heading3=heading3, path2r1=path2r1, path2r2=path2r2, path2l1=path2l1, path2l2=path2l2)
      return ret
    end

    # based on a Corner Homing 45 Cover pattern of touchpoints
    # this uses those touchpoints to create a representation of the corner in 3d robot space.
    def analyze_touchpoints_only_cover(p11, p12, p21, p3):
        zcoord=p3[2]

        # get the raw points from the first line
        l1p1x=p11[0]
        l1p1y=p11[1]
        l1p2x=p12[0]
        l1p2y=p12[1]

        # equate the first line in 2d space
        ml1 = (l1p2y-l1p1y) / (l1p2x-l1p1x)

        # b = y - mx
        bl1 = l1p1y - ml1 * l1p1x

        # get the raw points from the second line
        l2p1x=p21[0]
        l2p1y=p21[1]

        # equate the second line in 2d space
        # ml2 = opposite reciprocal of ml1 (because they are perpendicular) (assume perpendicular to make calculation of weldpath much easier)
        ml2 = -1 / ml1

        # b = y - mx
        bl2 = l2p1y - ml2 * l2p1x

        # find the intersection of the two lines
        # m1x+b1 = m2x+b2
        # m1x - m2x = b2 - b1
        # x = (b2-b1) / (m1-m2)
        xintersect = (bl2-bl1) / (ml1-ml2)
        yintersect = ml1 * xintersect + bl1

        pointintersect = p[xintersect,yintersect,zcoord,0,0,0]

        #FIND THE VECTORS
        #define a vector from the intersection to the second point on the first line
        l1delxfull = l1p2x - xintersect
        l1delyfull = l1p2y - yintersect

        l1delmag = sqrt(l1delxfull*l1delxfull + l1delyfull*l1delyfull)

        l1delxunit = l1delxfull / l1delmag
        l1delyunit = l1delyfull / l1delmag

        #define a vector from the intersection to the second point on the second line
        l2delxfull = l2p1x - xintersect
        l2delyfull = l2p1y - yintersect

        l2delmag = sqrt(l2delxfull*l2delxfull + l2delyfull*l2delyfull)

        l2delxunit = l2delxfull / l2delmag
        l2delyunit = l2delyfull / l2delmag

        #FIND HEADINGS
        #for each heading, find the angle of the line with respect to the pos x axis. this line is from pointintersect and along each edge of the corner
        heading1 = convert_uv_to_heading(l1delxunit, l1delyunit)
        heading3 = convert_uv_to_heading(l2delxunit, l2delyunit)
        # find halfway heading
        heading2 = (heading1 + heading3)/2

        #RETURN STRUCT
        ret = struct(pointintersect=pointintersect, heading1=heading1, heading2=heading2, heading3=heading3, l1delxunit=l1delxunit, l1delyunit=l1delyunit, l2delxunit=l2delxunit, l2delyunit=l2delyunit)
        return ret
    end

    # it takes 5 arguments as points
    # it returns a struct containing: (pointintersect, heading1, heading2, heading3, l1delxunit, l1delyunit, l2delxunit, l2delyunit)
    def analyze_touchpoints_only(p11, p12, p21, p22, p3):
      # FIND THE INTERSECTION
      # comment get the z
      zcoord=p3[2]

      # get the raw points from the first line
      l1p1x=p11[0]
      l1p1y=p11[1]
      l1p2x=p12[0]
      l1p2y=p12[1]

      # equate the first line in 2d space
      ml1 = (l1p2y-l1p1y) / (l1p2x-l1p1x)

      # b = y - mx
      bl1 = l1p1y - ml1 * l1p1x

      # get the raw points from the second line
      l2p1x=p21[0]
      l2p1y=p21[1]
      l2p2x=p22[0]
      l2p2y=p22[1]

      # equate the second line in 2d space
      ml2 = (l2p2y-l2p1y) / (l2p2x-l2p1x)

      # b = y - mx
      bl2 = l2p1y - ml2 * l2p1x


      # find the intersection of the two lines
      # m1x+b1 = m2x+b2
      # m1x - m2x = b2 - b1
      # x = (b2-b1) / (m1-m2)
      xintersect = (bl2-bl1) / (ml1-ml2)
      yintersect = ml1 * xintersect + bl1

      pointintersect = p[xintersect,yintersect,zcoord,0,0,0]

      #FIND THE VECTORS
      #define a vector from the intersection to the second point on the first line
      l1delxfull = l1p2x - xintersect
      l1delyfull = l1p2y - yintersect

      l1delmag = sqrt(l1delxfull*l1delxfull + l1delyfull*l1delyfull)

      l1delxunit = l1delxfull / l1delmag
      l1delyunit = l1delyfull / l1delmag

      #define a vector from the intersection to the second point on the second line
      l2delxfull = l2p2x - xintersect
      l2delyfull = l2p2y - yintersect

      l2delmag = sqrt(l2delxfull*l2delxfull + l2delyfull*l2delyfull)

      l2delxunit = l2delxfull / l2delmag
      l2delyunit = l2delyfull / l2delmag

      #FIND HEADINGS
      #for each heading, find the angle of the line with respect to the pos x axis. then add/subtract 90 degrees because you want to be perpendicular to that
      headingvector1 = convert_uv_to_heading(l1delxunit, l1delyunit)
      headingvector2 = convert_uv_to_heading(l2delxunit, l2delyunit)
      # find halfway heading
      heading2 = (headingvector1 + headingvector2)/2
      # find headings that the robot should face while traveling, perpendicular to the vectors of the sides of the box
      heading1 = headingvector1 + pi/2
      heading3 = headingvector2 - pi/2

      #RETURN STRUCT
      ret = struct(pointintersect=pointintersect, heading1=heading1, heading2=heading2, heading3=heading3, l1delxunit=l1delxunit, l1delyunit=l1delyunit, l2delxunit=l2delxunit, l2delyunit=l2delyunit)
      return ret
    end

    # given a struct from analyze_touchpoints_only(), calculate the points
    # for right, for non-extended
    def calculate_DOtA_points_right(struct1, listleans, chamferover):
        # get the stuff from the struct
        pointintersect = struct1[0]
        heading1 = struct1[1]
        heading2 = struct1[2]
        heading3 = struct1[3]
        l1delxunit = struct1[4]
        l1delyunit = struct1[5]
        l2delxunit = struct1[6]
        l2delyunit = struct1[7]

        # FIND THE POINTS ON THE LINES OF THE FIRST TURN PATH
        # find locations 8 inches away from  intersect point
        # CONST
        welddistance1 = 8 # vertical weld distance
        welddistance2 = 6 # first path second leg
        welddistance3 = 8 # second path second leg
        zup = .375
        # inches
        wd1 = welddistance1 * 25.4 / 1000
        wd2 = welddistance2 * 25.4 / 1000
        wd3 = welddistance3 * 25.4 / 1000
        zup = zup * 25.4 / 1000
        chamferovermm =  chamferover * 25.4 / 1000

        x = pointintersect[0] + l1delxunit * chamferovermm
        y = pointintersect[1] + l1delyunit * chamferovermm
        z = pointintersect[2] + zup

        #apply actual rxryrz to points
        # convert the headings to rxryrz and insert those values into the relevant points
        rxryrz = convert_heading_to_axang_preheatdown(heading1)
        rx = rxryrz[0]
        ry = rxryrz[1]
        rz = rxryrz[2]

        point1 = p[x + wd1*listleans[0], y + wd1*listleans[1], z + wd1, rx, ry, rz] # add in the listleans factor to follow the face of the box as we move up
        point2 = p[x, y, z, rx, ry, rz]

        # convert the headings to rxryrz and insert those values into the relevant points
        rxryrz = convert_heading_to_axang_ccw(heading1)
        rx = rxryrz[0]
        ry = rxryrz[1]
        rz = rxryrz[2]

        point4 = p[x, y, z, rx, ry, rz]
        x = x + l1delxunit * wd2
        y = y + l1delyunit * wd2
        point5 = p[x, y, z, rx, ry, rz]

        # FIND THE POINTS ON THE LINES OF THE SECOND AROUND PATH
        roundoverdistance = 0.05
        rod = roundoverdistance * 25.4 / 1000

        # now we have the unit vector. extend the weld distance from the intersection
        x = pointintersect[0] + l1delxunit * chamferovermm
        y = pointintersect[1] + l1delyunit * chamferovermm
        # convert the headings to rxryrz and insert those values into the relevant points
        rxryrz = convert_heading_to_axang(heading1)
        rx = rxryrz[0]
        ry = rxryrz[1]
        rz = rxryrz[2]
        point_1 = p[x, y, z, rx, ry, rz]

        x = pointintersect[0] + l1delxunit * rod
        y = pointintersect[1] + l1delyunit * rod
        point_2 = p[x, y, z, rx, ry, rz]

        # now we have the unit vector. extend the weld distance from the intersection
        x = pointintersect[0] + l2delxunit * wd3
        y = pointintersect[1] + l2delyunit * wd3
        # convert the headings to rxryrz and insert those values into the relevant points
        rxryrz = convert_heading_to_axang(heading3)
        rx = rxryrz[0]
        ry = rxryrz[1]
        rz = rxryrz[2]
        point_5 = p[x, y, z, rx, ry, rz]

        x = pointintersect[0] + l2delxunit * rod
        y = pointintersect[1] + l2delyunit * rod
        point_4 = p[x, y, z, rx, ry, rz]

        #FIND POINT 3
        # by calling analyze_touchpoints()
        atret = analyze_touchpoints(point_2, point_1, point_4, point_5, pointintersect)
        point_3 = atret[5]


        struct2 = struct(point1=point1, point2=point2, point4=point4, point5=point5, point_1=point_1, point_2=point_2, point_3=point_3, point_4=point_4, point_5=point_5)
        return struct2
    end

    # given a struct from analyze_touchpoints_only(), calculate the points
    # for left, for non-extended
    def calculate_DOtA_points_left(struct1, listleans, chamferover):
        # get the stuff from the struct
        pointintersect = struct1[0]
        heading1 = struct1[1]
        heading2 = struct1[2]
        heading3 = struct1[3]
        l1delxunit = struct1[4]
        l1delyunit = struct1[5]
        l2delxunit = struct1[6]
        l2delyunit = struct1[7]

        # FIND THE POINTS ON THE LINES OF THE FIRST TURN PATH
        # find locations 8 inches away from  intersect point
        # CONST
        welddistance1 = 8 # vertical weld distance
        welddistance2 = 6 # first path second leg
        welddistance3 = 8 # second path second leg
        zup = .375
        # inches
        wd1 = welddistance1 * 25.4 / 1000
        wd2 = welddistance2 * 25.4 / 1000
        wd3 = welddistance3 * 25.4 / 1000
        zup = zup * 25.4 / 1000
        chamferovermm =  chamferover * 25.4 / 1000

        x = pointintersect[0] + l2delxunit * chamferovermm
        y = pointintersect[1] + l2delyunit * chamferovermm
        z = pointintersect[2] + zup

        #apply actual rxryrz to points
        # convert the headings to rxryrz and insert those values into the relevant points
        rxryrz = convert_heading_to_axang_preheatdown(heading3)
        rx = rxryrz[0]
        ry = rxryrz[1]
        rz = rxryrz[2]

        point1 = p[x + wd1*listleans[0], y + wd1*listleans[1], z + wd1, rx, ry, rz]
        point2 = p[x, y, z, rx, ry, rz]

        # convert the headings to rxryrz and insert those values into the relevant points
        rxryrz = convert_heading_to_axang(heading3)
        rx = rxryrz[0]
        ry = rxryrz[1]
        rz = rxryrz[2]

        point4 = p[x, y, z, rx, ry, rz]
        x = x + l2delxunit * wd2
        y = y + l2delyunit * wd2
        point5 = p[x, y, z, rx, ry, rz]

        # FIND THE POINTS ON THE LINES OF THE SECOND AROUND PATH
        roundoverdistance = 0.05
        rod = roundoverdistance * 25.4 / 1000

        # now we have the unit vector. extend the weld distance from the intersection
        x = pointintersect[0] + l2delxunit * chamferovermm
        y = pointintersect[1] + l2delyunit * chamferovermm
        # convert the headings to rxryrz and insert those values into the relevant points
        rxryrz = convert_heading_to_axang_ccw(heading3)
        rx = rxryrz[0]
        ry = rxryrz[1]
        rz = rxryrz[2]
        point_1 = p[x, y, z, rx, ry, rz]

        x = pointintersect[0] + l2delxunit * rod
        y = pointintersect[1] + l2delyunit * rod
        point_2 = p[x, y, z, rx, ry, rz]

        # now we have the unit vector. extend the weld distance from the intersection
        x = pointintersect[0] + l1delxunit * wd3
        y = pointintersect[1] + l1delyunit * wd3
        # convert the headings to rxryrz and insert those values into the relevant points
        rxryrz = convert_heading_to_axang_ccw(heading1)
        rx = rxryrz[0]
        ry = rxryrz[1]
        rz = rxryrz[2]
        point_5 = p[x, y, z, rx, ry, rz]

        x = pointintersect[0] + l1delxunit * rod
        y = pointintersect[1] + l1delyunit * rod
        point_4 = p[x, y, z, rx, ry, rz]

        #FIND POINT 3
        # by calling analyze_touchpoints()
        atret = analyze_touchpoints(point_2, point_1, point_4, point_5, pointintersect)
        point_3 = atret[5]
        #point 3 will not have the correct rxryrz though because now the gun needs to be face up.
        rxryrz = convert_heading_to_axang_ccw(heading2)
        rx = rxryrz[0]
        ry = rxryrz[1]
        rz = rxryrz[2]
        point_3 = p[point_3[0], point_3[1], point_3[2], rx, ry, rz]

        struct2 = struct(point1=point1, point2=point2, point4=point4, point5=point5, point_1=point_1, point_2=point_2, point_3=point_3, point_4=point_4, point_5=point_5)
        return struct2
    end

    # given a struct from analyze_touchpoints_only(), calculate the points
    # for right, for extended
    def calculate_DOtA_points_right_extended(struct1, listleans, chamferover, chamferup, tcp_pose_top):
        # get the stuff from the struct
        pointintersect = struct1[0]
        heading1 = struct1[1]
        heading2 = struct1[2]
        heading3 = struct1[3]
        l1delxunit = struct1[4]
        l1delyunit = struct1[5]
        l2delxunit = struct1[6]
        l2delyunit = struct1[7]

        # FIND THE POINTS ON THE LINES OF THE FIRST TURN PATH
        # find locations 8 inches away from  intersect point
        # CONST
        # welddistance1 = 8 # vertical weld distance
        welddistance2 = 5 # first path second leg
        welddistance3 = 5 # second path second leg

        # inches
        # wd1 = welddistance1 * 25.4 / 1000
        wd2 = welddistance2 * 25.4 / 1000
        wd3 = welddistance3 * 25.4 / 1000
        zup = chamferup * 25.4 / 1000
        chamferovermm =  chamferover * 25.4 / 1000

        # weld distance is the distance that it will weld. this will make it start at the z height that the user specified
        wd1 = tcp_pose_top[2] - pointintersect[2] - zup

        x = pointintersect[0] + l1delxunit * chamferovermm
        y = pointintersect[1] + l1delyunit * chamferovermm
        z = pointintersect[2] + zup

        #apply actual rxryrz to points
        # convert the headings to rxryrz and insert those values into the relevant points
        rxryrz = convert_heading_to_axang_preheatdown(heading1)
        rx = rxryrz[0]
        ry = rxryrz[1]
        rz = rxryrz[2]

        point1 = p[x + wd1*listleans[0], y + wd1*listleans[1], z + wd1, rx, ry, rz] # add in the listleans factor to follow the face of the box as we move up
        point2 = p[x, y, z, rx, ry, rz]

        # convert the headings to rxryrz and insert those values into the relevant points
        rxryrz = convert_heading_to_axang_ccw(heading1)
        rx = rxryrz[0]
        ry = rxryrz[1]
        rz = rxryrz[2]

        point4 = p[x, y, z, rx, ry, rz]
        x = x + l1delxunit * wd2
        y = y + l1delyunit * wd2
        point5 = p[x, y, z, rx, ry, rz]

        # FIND THE POINTS ON THE LINES OF THE SECOND AROUND PATH
        roundoverdistance = 0.05
        rod = roundoverdistance * 25.4 / 1000

        # now we have the unit vector. extend the weld distance from the intersection
        x = pointintersect[0] + l1delxunit * chamferovermm
        y = pointintersect[1] + l1delyunit * chamferovermm
        # convert the headings to rxryrz and insert those values into the relevant points
        rxryrz = convert_heading_to_axang(heading1)
        rx = rxryrz[0]
        ry = rxryrz[1]
        rz = rxryrz[2]
        point_1 = p[x, y, z, rx, ry, rz]

        x = pointintersect[0] + l1delxunit * rod
        y = pointintersect[1] + l1delyunit * rod
        point_2 = p[x, y, z, rx, ry, rz]

        # convert the headings to rxryrz and insert those values into the relevant points
        rxryrz = convert_heading_to_axang(heading3)
        rx = rxryrz[0]
        ry = rxryrz[1]
        rz = rxryrz[2]

        x = pointintersect[0] + l2delxunit * rod
        y = pointintersect[1] + l2delyunit * rod
        point_4 = p[x, y, z, rx, ry, rz]

        # now we have the unit vector. extend the weld distance from the intersection
        x = pointintersect[0] + l2delxunit * wd3
        y = pointintersect[1] + l2delyunit * wd3
        point_5 = p[x, y, z, rx, ry, rz]

        #FIND POINT 3
        # by calling analyze_touchpoints()
        atret = analyze_touchpoints(point_2, point_1, point_4, point_5, pointintersect)
        atret5 = atret[5]
        point_3 = p[atret5[0], atret5[1], z, atret5[3], atret5[4], atret5[5]]


        struct2 = struct(point1=point1, point2=point2, point4=point4, point5=point5, point_1=point_1, point_2=point_2, point_3=point_3, point_4=point_4, point_5=point_5)
        return struct2
    end

    # given a struct from analyze_touchpoints_only(), calculate the points
    # for left, for extended
    def calculate_DOtA_points_left_extended(struct1, listleans, chamferover, chamferup, tcp_pose_top):
        # get the stuff from the struct
        pointintersect = struct1[0]
        heading1 = struct1[1]
        heading2 = struct1[2]
        heading3 = struct1[3]
        l1delxunit = struct1[4]
        l1delyunit = struct1[5]
        l2delxunit = struct1[6]
        l2delyunit = struct1[7]

        # FIND THE POINTS ON THE LINES OF THE FIRST TURN PATH
        # find locations 8 inches away from  intersect point
        # CONST
        # welddistance1 = 8 # vertical weld distance
        welddistance2 = 5 # first path second leg
        welddistance3 = 5 # second path second leg

        # inches
        # wd1 = welddistance1 * 25.4 / 1000
        wd2 = welddistance2 * 25.4 / 1000
        wd3 = welddistance3 * 25.4 / 1000
        zup = chamferup * 25.4 / 1000
        chamferovermm =  chamferover * 25.4 / 1000

        # weld distance is the distance that it will weld. this will make it start at the z height that the user specified
        wd1 = tcp_pose_top[2] - pointintersect[2] - zup

        x = pointintersect[0] + l2delxunit * chamferovermm
        y = pointintersect[1] + l2delyunit * chamferovermm
        z = pointintersect[2] + zup

        #apply actual rxryrz to points
        # convert the headings to rxryrz and insert those values into the relevant points
        rxryrz = convert_heading_to_axang_preheatdown(heading3)
        rx = rxryrz[0]
        ry = rxryrz[1]
        rz = rxryrz[2]

        point1 = p[x + wd1*listleans[0], y + wd1*listleans[1], z + wd1, rx, ry, rz]
        point2 = p[x, y, z, rx, ry, rz]

        # convert the headings to rxryrz and insert those values into the relevant points
        rxryrz = convert_heading_to_axang(heading3)
        rx = rxryrz[0]
        ry = rxryrz[1]
        rz = rxryrz[2]

        point4 = p[x, y, z, rx, ry, rz]
        x = x + l2delxunit * wd2
        y = y + l2delyunit * wd2
        point5 = p[x, y, z, rx, ry, rz]

        # FIND THE POINTS ON THE LINES OF THE SECOND AROUND PATH
        roundoverdistance = 0.05
        rod = roundoverdistance * 25.4 / 1000

        # now we have the unit vector. extend the weld distance from the intersection
        x = pointintersect[0] + l2delxunit * chamferovermm
        y = pointintersect[1] + l2delyunit * chamferovermm
        # convert the headings to rxryrz and insert those values into the relevant points
        rxryrz = convert_heading_to_axang_ccw(heading3)
        rx = rxryrz[0]
        ry = rxryrz[1]
        rz = rxryrz[2]
        point_1 = p[x, y, z, rx, ry, rz]

        x = pointintersect[0] + l2delxunit * rod
        y = pointintersect[1] + l2delyunit * rod
        point_2 = p[x, y, z, rx, ry, rz]

        # convert the headings to rxryrz and insert those values into the relevant points
        rxryrz = convert_heading_to_axang_ccw(heading1)
        rx = rxryrz[0]
        ry = rxryrz[1]
        rz = rxryrz[2]

        x = pointintersect[0] + l1delxunit * rod
        y = pointintersect[1] + l1delyunit * rod
        point_4 = p[x, y, z, rx, ry, rz]

        # now we have the unit vector. extend the weld distance from the intersection
        x = pointintersect[0] + l1delxunit * wd3
        y = pointintersect[1] + l1delyunit * wd3
        point_5 = p[x, y, z, rx, ry, rz]

        #FIND POINT 3
        # by calling analyze_touchpoints()
        atret = analyze_touchpoints(point_2, point_1, point_4, point_5, pointintersect)
        point_3 = atret[5]
        #point 3 will not have the correct rxryrz though because now the gun needs to be face up
        rxryrz = convert_heading_to_axang_ccw(heading2)
        rx = rxryrz[0]
        ry = rxryrz[1]
        rz = rxryrz[2]
        point_3 = p[point_3[0], point_3[1], z, rx, ry, rz]

        struct2 = struct(point1=point1, point2=point2, point4=point4, point5=point5, point_1=point_1, point_2=point_2, point_3=point_3, point_4=point_4, point_5=point_5)
        return struct2
    end

    # this function analyzes the vertical points
    # calculates the slope of the edge in question
    # specifically, for each inch up in the z direction, what is the change in x and change in y direction
    # returns a list of [nx, ny]
    def analyze_vertical_touchpoints(p11, p12, p13, p21, p22, p23, p3):
        # first, find the equations of the planes from the 6 points
        plane1 = findplane(p11, p12, p13)
        plane2 = findplane(p21, p22, p23)
        # Find the Direction Vector of the Line: The direction vector d of the line of intersection can be found by taking the cross product of the normal vectors of each plane (a, b, and c)
        nx = plane1[1]*plane2[2] - plane1[2]*plane2[1]
        ny = plane1[2]*plane2[0] - plane1[0]*plane2[2]
        nz = plane1[0]*plane2[1] - plane1[1]*plane2[0]
        # normalize the vector so the z length is 1
        multiplier = 1 / nz
        nx = nx * multiplier
        ny = ny * multiplier
        nz = nz * multiplier # should become equal to 1
        ret = [nx, ny]
        return ret
    end

    # given 3 points, this finds the plane and its equation
    # rereturns ax + by + cz + d = 0 in a list of [a, b, c, d]
    def findplane(p11, p12, p13):
        # extract coordinates
        x1 = p11[0]
        y1 = p11[1]
        z1 = p11[2]
        x2 = p12[0]
        y2 = p12[1]
        z2 = p12[2]
        x3 = p13[0]
        y3 = p13[1]
        z3 = p13[2]
        # create vectors from the points
        v1x = x2-x1
        v1y = y2-y1
        v1z = z2-z1
        v2x = x3-x1
        v2y = y3-y1
        v2z = z3-z1
        #calculate the normal vector using the cross product
        nx = v1y*v2z - v1z*v2y # i component
        ny = v1z*v2x - v1x*v2z # j component
        nz = v1x*v2y - v1y*v2x # k component
        # calculate d in the plane equation
        d = -1 * (nx*x1 + ny*y1 + nz*z1)
        ret = [nx, ny, nz, d]
        return ret
    end

    # given a heading, (ccw from +x axis), find the mx+b slope
    # fails if exactly vertical
    def get_slope_from_heading(heading):
        return tan(heading)
    end



    # this function finds the points (and rxryrz) of the 2 points (start and end) of vertical weld section
    def find_vertical_points(pointintersect, l1delxunit, l1delyunit, l2delxunit, l2delyunit, offset, wd, heading1, heading3):

      # find right side stuff
      # find the point in 3d space that is .375 up and .375 over
      x = pointintersect[0] + l1delxunit * offset
      y = pointintersect[1] + l1delyunit * offset
      z = pointintersect[2] + offset
      # find rxryrz
      rxryrz = convert_heading_to_axang_preheatup(heading1)
      rx = rxryrz[0]
      ry = rxryrz[1]
      rz = rxryrz[2]
      path2r1 = p[x, y, z, rx, ry, rz]
      path2r2 = p[x, y, z + wd, rx, ry, rz]

      # find left side
      # find the point in 3d space that is .375 up and .375 over
      x = pointintersect[0] + l2delxunit * offset
      y = pointintersect[1] + l2delyunit * offset
      z = pointintersect[2] + offset
      # find rxryrz
      rxryrz = convert_heading_to_axang_preheatup(heading3)
      rx = rxryrz[0]
      ry = rxryrz[1]
      rz = rxryrz[2]
      path2l1 = p[x, y, z, rx, ry, rz]
      path2l2 = p[x, y, z + wd, rx, ry, rz]

      ret = struct(path2r1=path2r1, path2r2=path2r2, path2l1=path2l1, path2l2=path2l2)
      return ret
    end

    # this function converts a unit vector to its heading angle ccw from x+ axis
    # takes uvx and uvy
    # returns heading in radians
    def convert_uv_to_heading(uvx, uvy):
      baseang = atan(uvy/uvx)
      if uvx < 0:
        ang = baseang + pi
      elif uvy < 0:
        ang = baseang + pi * 2
      else:
        ang = baseang
      end
      return ang
    end

    # this function finds the equation of a line, perpendicular to a given line, and going through a given point
    # takes 3 arguments: m (the original line's slope), x (point's x coord), y (point's y coord). the b of the original line is not needed
    # returns a list of [m,b] (the slope and intercept of the new line)
    def find_perpendicular_line(origm, x, y):
      m = (1/origm) * -1
      b = y - m*x
      ret = [m, b]
      return ret
    end

    # this function finds the intersection point between two lines in the xy plane
    # takes 4 arguments: m1, b1, m2, b2
    # returns a list of [x,y] (the point of intersection)
    def find_intersection(m1, b1, m2, b2):
      # m1x+b1 = m2x+b2
      # m1x - m2x = b2 - b1
      # x = (b2-b1) / (m1-m2)
      x = (b2-b1) / (m1-m2)
      y = m1 * x + b1
      ret = [x, y]
      return ret
    end

    # this function finds the distance between 2 points in 3d space
    # it takes 6 arguments: x1, y1, z1, x2, y2, z2
    # it returns a distance
    def distance_between(x1, y1, z1, x2, y2, z2):
      distsquared = (x2-x1)*(x2-x1)+(y2-y1)*(y2-y1)+(z2-z1)*(z2-z1)
      dist = sqrt(distsquared)
      return dist
    end

    # this function takes a point, a unit vector, and a distance, and adds the distance to the point in the direction of the unit vector (3d space)
    # it returns a point as a list of coordinates
    def add_vectordistance_to_point(xi, yi, zi, uvx, uvy, uvz, delta):
      xf = xi + uvx * delta
      yf = yi + uvy * delta
      zf = zi + uvz * delta
      ret = [xf, yf, zf]
      return ret
    end

    # this function converts a heading (ccw radians from the positive x axis) into rxryrz to be put into a point p[]
    # this will point the gun in this heading with the bottom side of the gun facing up.
    # the values used in this program were calculated by doing rotation matrix math in the file on WI-CALVINB10 C. Documents. Theory for converting rotations into axis angle representations
    def convert_heading_to_axang(heading):
     axisxraw = -1 * sin(heading)
     axisyraw = cos(heading) + 1
     axiszraw = sin(heading)

     magnitude = sqrt(axisxraw*axisxraw + axisyraw*axisyraw + axiszraw*axiszraw)

     axisxunit = axisxraw / magnitude
     axisyunit = axisyraw / magnitude
     axiszunit = axiszraw / magnitude

     angle = acos( (cos(heading) - 1) / 2 )

     rxout = axisxunit * angle
     ryout = axisyunit * angle
     rzout = axiszunit * angle

     return [rxout, ryout, rzout]
    end

    # this function converts a heading (ccw radians from the positive x axis) into rxryrz to be put into a point p[]
    # this will point the gun in this heading with the preheat side of the gun tip facing up. Used for welding in a vertical path.
    # the values used in this program were calculated by doing rotation matrix math in the file on WI-CALVINB10 C. Documents. Theory for converting rotations into axis angle representations
    def convert_heading_to_axang_preheatup(heading):
     axisxraw = -sin(heading) + 1
     axisyraw = cos(heading)
     axiszraw = cos(heading)

     magnitude = sqrt(axisxraw*axisxraw + axisyraw*axisyraw + axiszraw*axiszraw)

     axisxunit = axisxraw / magnitude
     axisyunit = axisyraw / magnitude
     axiszunit = axiszraw / magnitude

     angle = acos( (-sin(heading) - 1) / 2 )

     rxout = axisxunit * angle
     ryout = axisyunit * angle
     rzout = axiszunit * angle

     return [rxout, ryout, rzout]
    end

    # this function converts a heading (ccw radians from the positive x axis) into rxryrz to be put into a point p[]
    # this will point the gun in this heading with the preheat side of the gun tip facing down. Used for welding in a vertical path downwards.
    # the values used in this program were calculated by doing rotation matrix math in the file on WI-CALVINB10 C. Documents. Theory for converting rotations into axis angle representations
    def convert_heading_to_axang_preheatdown(heading):
     axisxraw = -sin(heading) - 1
     axisyraw = cos(heading)
     axiszraw = -cos(heading)

     magnitude = sqrt(axisxraw*axisxraw + axisyraw*axisyraw + axiszraw*axiszraw)

     axisxunit = axisxraw / magnitude
     axisyunit = axisyraw / magnitude
     axiszunit = axiszraw / magnitude

     angle = acos( (sin(heading) - 1) / 2 )

     rxout = axisxunit * angle
     ryout = axisyunit * angle
     rzout = axiszunit * angle

     return [rxout, ryout, rzout]
    end

    # this function converts a heading (ccw radians from the positive x axis) into rxryrz to be put into a point p[]
    # this will point the gun in this heading with the preheat side of the gun tip facing right. Used for welding counterclockwise around the box.
    # the values used in this program were calculated by doing rotation matrix math in the file on WI-CALVINB10 C. Documents. Theory for converting rotations into axis angle representations
    def convert_heading_to_axang_ccw(heading):
     axisxraw = -sin(heading)
     axisyraw = cos(heading) - 1
     axiszraw = -sin(heading)

     magnitude = sqrt(axisxraw*axisxraw + axisyraw*axisyraw + axiszraw*axiszraw)

     axisxunit = axisxraw / magnitude
     axisyunit = axisyraw / magnitude
     axiszunit = axiszraw / magnitude

     angle = acos( (-cos(heading) - 1) / 2 )

     rxout = axisxunit * angle
     ryout = axisyunit * angle
     rzout = axiszunit * angle

     return [rxout, ryout, rzout]
    end

    # this function is for getting the points along the path of the corner homing 45
    # point0 is the point where they touched
    def get_corner_homing_45_pathpoints(point0, pointtop = p[0,0,0,0,0,0]):
      p0x = point0[0]
      p0y = point0[1]
      p0z = point0[2]
      p0rx = point0[3]
      p0ry = point0[4]
      p0rz = point0[5]

      #constants
      #distances of how far away from point the touchpoints are
      d0 = 0.10 # how far from the box to retreat and approach
      d1 = 0.06 # first distance from init point
      d2 = 0.15 # second distance from init point
      d3 = 0.125 #vertical distance from first point
      sqrt2 = 0.707106781 # 1/sqrt(2) , the inverse of the sqrt(2)

      ph1 = p[p0x + d0, p0y, p0z + d1, p0rx, p0ry, p0rz] #approach point for turn

      ph2 = p[p0x+d0-d0*0.5-sqrt2*d1, p0y+d0*0.5+sqrt2*d1, p0z+d1, 1.446, -0.8, -0.733]
      ph3 = p[p0x+d0-d0*0.5-sqrt2*d2, p0y+d0*0.5+sqrt2*d2, p0z+d1, 1.446, -0.8, -0.733]
      ph4 = p[p0x+d0-d0*0.5-sqrt2*d1, p0y-d0*0.5-sqrt2*d1, p0z+d1, 0.626, -1.993, -1.813]
      ph5 = p[p0x+d0-d0*0.5-sqrt2*d2, p0y-d0*0.5-sqrt2*d2, p0z+d1, 0.626, -1.993, -1.813]

      # go back to ph1
      ph6 = p[p0x + d0, p0y, p0z -0.05, 0, 0, pi] # approach point for under turn
      # moveL from ph1 to ph6
      ph7 = p[p0x-d1, p0y, p0z-0.05, 0, 0, pi]

      # add the vertical touch points
      if pointtop[2] == 0:
        ph2up = p[ph2[0], ph2[1], ph2[2]+d3, ph2[3], ph2[4], ph2[5]]
        ph4up = p[ph4[0], ph4[1], ph4[2]+d3, ph4[3], ph4[4], ph4[5]]
      elif pointtop[2] > p0z + 0.914: # 0.914m = 36 inches
        ph2up = p[ph2[0], ph2[1], p0z + 0.914, ph2[3], ph2[4], ph2[5]]
        ph4up = p[ph4[0], ph4[1], p0z + 0.914, ph4[3], ph4[4], ph4[5]]
      else:
        ph2up = p[ph2[0], ph2[1], pointtop[2], ph2[3], ph2[4], ph2[5]]
        ph4up = p[ph4[0], ph4[1], pointtop[2], ph4[3], ph4[4], ph4[5]]
      end
      ret = struct(ph1=ph1, ph2=ph2, ph3=ph3, ph4=ph4, ph5=ph5, ph6=ph6, ph7=ph7, ph2up=ph2up, ph4up=ph4up)
      is_robot_at_reachable_spot(point0, ret)
      return ret
    end

    def get_corner_homing_45_pathpoints_cover(point0):
        p0x = point0[0]
        p0y = point0[1]
        p0z = point0[2]
        p0rx = point0[3]
        p0ry = point0[4]
        p0rz = point0[5]

        #constants
        #distances of how far away from point the touchpoints are
        d0 = 0.10 # how far from the box to retreat and approach
        d1 = 0.04 # first distance from init point
        d2 = 0.15 # second distance from init point
        d4 = 0.06 # top distance from init point - larger to avoid large chamfers
        sqrt2 = 0.707106781 # 1/sqrt(2) , the inverse of the sqrt(2)

        ph1 = p[p0x + d0, p0y, p0z + d1, p0rx, p0ry, p0rz] #approach point for turn

        ph2 = p[p0x+d0-d0*0.5-sqrt2*d1, p0y+d0*0.5+sqrt2*d1, p0z-d1, 1.446, -0.8, -0.733]
        ph3 = p[p0x+d0-d0*0.5-sqrt2*d2, p0y+d0*0.5+sqrt2*d2, p0z-d1, 1.446, -0.8, -0.733]
        ph4 = p[p0x+d0-d0*0.5-sqrt2*d1, p0y-d0*0.5-sqrt2*d1, p0z-d1, 0.626, -1.993, -1.813]
        #ph5 = p[p0x+d0-d0*0.5-sqrt2*d2, p0y-d0*0.5-sqrt2*d2, p0z-d1, 0.626, -1.993, -1.813]

        # approach point for top
        ph6 = p[p0x + d0 * 2, p0y, p0z+0.05, 0.138, 3.104, -0.072] # double the d0 in the x direction because it was getting VERY close to smacking the corner.

        # top point
        ph7 = p[p0x - d4, p0y, p0z+0.05, 0.138, 3.104, -0.072]

        ret = struct(ph1=ph1, ph2=ph2, ph3=ph3, ph4=ph4, ph5=ph4, ph6=ph6, ph7=ph7)
        is_robot_at_reachable_spot(point0, ret)
        return ret
    end

    # this function determines the starting touchpoints for homing in on cover straight geometry
    # includes two side points to determine the sidewall plane (assumed vertical) and two top points to determine top plane (assumed perpendicular to sidewall plane)
    def get_straight_homing_pathpoints_cover(leftpoint, rightpoint):
        # get the teach position points
        lpx = leftpoint[0]
        lpy = leftpoint[1]
        lpz = leftpoint[2]
        rpx = rightpoint[0]
        rpy = rightpoint[1]
        rpz = rightpoint[2]

        # specify the distances from
        d0 = 0.05 # how far from the planes to approach from
        d1 = 0.03 # how far from the teach point to home from, when there is no chamfer to avoid
        d2 = 0.06 # how far from the teach point to home from, when there is a chamfer to avoid

        # calculate the points (the rxryrz are given in pretend_welder_top coordinates. they match pure rotations of 90 degrees)
        ph1 = p[lpx + d0, lpy, lpz - d1, 1.209, -1.209, -1.209] # left side approach
        ph2 = p[rpx + d0, rpy, rpz - d1, 1.209, -1.209, -1.209] # right side approach
        ph3 = p[lpx - d2, lpy, lpz + d0, 2.221, -2.221, 0] # left top approach
        ph4 = p[rpx - d2, rpy, rpz + d0, 2.221, -2.221, 0] # right top approach

        ret = struct(ph1=ph1, ph2=ph2, ph3=ph3, ph4=ph4)
        is_robot_at_reachable_spot(leftpoint, ret)
        return ret
    end

    # this function determines the starting touchpoints for homing in on cover straight geometry
    # includes two side points to determine the sidewall plane (assumed vertical) and two top points to determine top plane (assumed perpendicular to sidewall plane)
    def get_straight_homing_pathpoints_floor(leftpoint, rightpoint):
        # get the teach position points
        lpx = leftpoint[0]
        lpy = leftpoint[1]
        lpz = leftpoint[2]
        rpx = rightpoint[0]
        rpy = rightpoint[1]
        rpz = rightpoint[2]

        # specify the distances from
        d0 = 0.05 # how far from the planes to approach from
        d1 = 0.03 # how far from the teach point to home from, when there is no chamfer to avoid
        d2 = 0.06 # how far from the teach point to home from, when there is a chamfer to avoid

        # calculate the points
        ph1 = p[lpx + d0, lpy, lpz + d1, 1.209, -1.209, -1.209] # left side approach
        ph2 = p[rpx + d0, rpy, rpz + d1, 1.209, -1.209, -1.209] # right side approach
        ph3 = p[lpx - d1, lpy, lpz - d0, 0, 0, 0] # left bottom approach
        ph4 = p[rpx - d1, rpy, rpz - d0, 0, 0, 0] # right bottom approach

        ret = struct(ph1=ph1, ph2=ph2, ph3=ph3, ph4=ph4)
        is_robot_at_reachable_spot(leftpoint, ret, 4)
        return ret
    end

    # this function checks whether the touchpoints are reachable AKA is the robot positioned in the right spot
    # if everything looks good, it continues.
    # if it detects a problem, it infinite loops a popup
    def is_robot_at_reachable_spot(point0, struct_touchpoints, structlength = 9):
      # first, check whether the corner is too low to the ground that the bottom homing will hit the ground (z < -400)
      lc_height = get_lift_column_height_condensed()
      # total height = zeroed lift column height (41.25 inches) (1.04775 m) plus lift column height plus robot relative height
      totalheight = 1.04775 + lc_height + point0[2]
      if totalheight < 1.04775 - 0.400:
        # bad
        popuptext = "Tank Corner is too low to the ground. Collisions will occur. Stop Program and raise tank. "
        # infinite loop
        while 1==1:
          popup(popuptext, title="Robot Positioning Warning",blocking=True)
        end
      end



      # next, check whether the touchpoints are reachable
      allvalid = check_structofpoints_validity(struct_touchpoints)
      if not allvalid:

        # then unreachable
        # generate message
        listproblems = ""
        listnames = ["ph1", "ph2", "ph3", "ph4", "ph5", "ph6", "ph7", "ph2up", "ph4up"]
        i = 0
        # structlength = 9 # used to be a declare statement here. now it is a parameter. floor corner has 9. other features have less
        while i < structlength:
          curr = struct_touchpoints[i]
          valid = get_inverse_kin_has_solution(curr)
          if not valid:
            listproblems = listproblems + listnames[i]
          end
          i = i + 1
        end
        # display
        popuptext = "Robot is too far from tank corner. Cannot reach some necessary positions. Stop Program and move robot closer. " + listproblems
        # infinite loop
        while 1==1:
          popup(popuptext, title="Robot Positioning Warning",blocking=True)
        end
      end

    end

    # this function takes a struct of points as an argument, and checks whether every point in the list is reachable using get_inverse_kin_has_solution()
    # this function does NOT check for weird twists or joint limits
    # inputstruct must contain only points
    # it returns true if all points are valid. it returns false if any points are valid
    # a list of length 0 indicates that all points are valid
    def check_structofpoints_validity(inputstruct):
      # next, check whether the touchpoints are reachable
      structlength = length(inputstruct)
      i = 0
      allvalid = True
      while i < structlength:
        curr = inputstruct[i]
        valid = get_inverse_kin_has_solution(curr)
        if not valid:
          return False
        end
        i = i + 1
      end
      return True
    end

    # checks the validity of all points during a left weld
    # takes 2 arguments: struct1 (struct1[0] has to contain pointintersect) and struct2 (contains all the points (9) of the weld path)
    def check_validity_left(struct1, struct2):
      #first, check whether robot is too close
      pointintersect = struct1[0]
      # next, check if the corner is too close to the robot to do a left around weld (complex but approximately X > -1300)
      # if y < 0, then x < -1300. if y < 480, then y > (1300+x)*8. if y > 480, then y > (1235+x)*4 + 500
      toocloseleftweld = False
      if pointintersect[1] < 0:
        if pointintersect[0] > -1.300:
          toocloseleftweld = True
        end
      elif pointintersect[1] < 0.480:
        if pointintersect[1] < (1.300 + pointintersect[0])*8:
          toocloseleftweld = True
        end
      else:
        if pointintersect[1] < (1.235 + pointintersect[0])*4 + 0.500:
          toocloseleftweld = True
        end
      end
      if toocloseleftweld:
        # bad
        popuptext = "Robot is too close to tank corner. Collisions may occur. Stop Program and move robot farther. "
        # infinite loop
        while 1==1:
          popup(popuptext, title="Robot Positioning Warning",blocking=True)
        end
      end

      #next, check whether all the points in the weldpath are valid
      structlength = 9
      i = 0
      allvalid = True
      listproblems = ""
      listnames = ["point1", "point2", "point4", "point5", "point_1", "point_2", "point_3", "point_4", "point_5"]
      while i < structlength:
        curr = struct2[i]
        valid = get_inverse_kin_has_solution(curr)
        if not valid:
          if i > 0:
            allvalid = False
            listproblems = listproblems + listnames[i]
          end
        end
        i = i + 1
      end

      if not allvalid:
        # display
        popuptext = "Robot is too far from tank corner. Cannot reach some necessary positions. Stop Program and move robot closer. " + listproblems
        # infinite loop
        while 1==1:
          popup(popuptext, title="Robot Positioning Warning",blocking=True)
        end
      end

      # check whether the path involves weird turns or joint limits. currently just checks the first position
      p_prev = [-0.021118, -1.26292, 2.43578, 5.07088, -2.29912, 1.53362] #last point of left weld prerotate
      joints_1 = get_inverse_kin(struct2[0], p_prev) # struct2[0] is point1
      allGood = True
      i = 0
      structlength = 6
      while i < structlength:
        joint_curr = joints_1[i]
        # check for anything that exceeds joint limits
        degreesmax = 360 * pi / 180
        if joint_curr > degreesmax or joint_curr < degreesmax * -1:
          allGood = False
        end
        # check for anything that is significantly different than the aligned approach. could indicate a twist is needed. we dont want that
        maxdifference = 150 * pi / 180
        difference = joint_curr - p_prev[i]
        if difference > maxdifference or difference * -1 > maxdifference:
          allGood = False
        end
        i = i + 1
      end

      if not allGood:
        # call lift column extend function
        struct2 = floor_corner_lift_column_extend_left(struct2)

      end

      # return struct2 back
      return struct2
    end

    # checks the validity of all points during a right weld
    def check_validity_right(struct1, struct2):
      # first, check whether the right pivot will bonk itself
      pointintersect = struct1[0]
      heading1 = struct1[1] # this is the direction that the welder will face when doing the right side of the box

      #first, check whether the heading is just too far offset
      # more than 15 degrees off of 45 is too much
      # normal heading is 216 degrees
      #201 degrees to 231 degrees
      heading1degrees = heading1 * 180 / pi
      if heading1degrees < 201 or heading1degrees > 231 :
        # then out of range
        popuptext = "Robot is not aligned at a 45 degree angle of corner (15 degree leeway). Collisions may occur. Stop Program and align robot. heading1degrees=" + str_cat("",heading1degrees)
        # infinite loop
        while 1==1:
          popup(popuptext, title="Robot Positioning Warning",blocking=True)
        end
      end

      #TODO: add the checks for whether x is too close, given the heading
      # add checks for whether x is too close, given the heading
      # different equations for whether heading offset > 5 degrees or less (inc. negative)
      headingoffset = heading1degrees - 216
      if headingoffset < 5:
        # then calculate a and b
        a = 0.4584 + -0.02369 * headingoffset
        b = (-1151.4 + 13.83 * headingoffset) / 1000
        # check whether x > a*y+b
        if pointintersect[0] > a * pointintersect[1] + b:
          # bad
          popuptext = "Robot is too close to tank corner or not at the right angle. Collisions may occur. Stop Program and align robot. "
          # infinite loop
          while 1==1:
            popup(popuptext, title="Robot Positioning Warning",blocking=True)
          end
        end
      else:
        # headingoffset > 5 degrees
        if pointintersect[1] < 0:
          if pointintersect[0] > -1150.0 / 1000.0:
            #bad
            popuptext = "Robot is too close to tank corner. Collisions may occur. Stop Program and align robot. "
            # infinite loop
            while 1==1:
              popup(popuptext, title="Robot Positioning Warning",blocking=True)
            end
          end
        else:
          # if x > .7736 y - 1101.9 then bad
          if pointintersect[0] > 0.7736 * pointintersect[1] - 1101.9 / 1000:
            popuptext = "Robot is too close to tank corner. Collisions may occur. Stop Program and align robot. "
            # infinite loop
            while 1==1:
              popup(popuptext, title="Robot Positioning Warning",blocking=True)
            end
          end
        end
      end

      #next, check whether all the points in the weldpath are valid
      structlength = 9
      i = 0
      allvalid = True
      listproblems = ""
      listnames = ["point1", "point2", "point4", "point5", "point_1", "point_2", "point_3", "point_4", "point_5"]
      while i < structlength:
        curr = struct2[i]
        valid = get_inverse_kin_has_solution(curr)
        if not valid:
          if i > 0:
            allvalid = False
            listproblems = listproblems + listnames[i]
          end
        end
        i = i + 1
      end

      if not allvalid:
        # display
        popuptext = "Robot is too far from tank corner. Cannot reach some necessary positions. Stop Program and move robot closer. " + listproblems
        # infinite loop
        while 1==1:
          popup(popuptext, title="Robot Positioning Warning",blocking=True)
        end
      end

      # check whether the path involves weird turns or joint limits. first position
      p_prev = [-1.13307, -1.48911, 2.84785, 4.92357, -4.89059, 1.57184] #last point of right weld prerotate
      joints_1 = get_inverse_kin(struct2[0], p_prev) # struct2[0] is point1
      allGood = True
      i = 0
      structlength = 6
      while i < structlength:
        joint_curr = joints_1[i]
        # check for anything that exceeds joint limits
        degreesmax = 360 * pi / 180
        if joint_curr > degreesmax or joint_curr < degreesmax * -1:
          allGood = False
        end
        # check for anything that is significantly different than the aligned approach. could indicate a twist is needed. we dont want that
        maxdifference = 150 * pi / 180
        difference = joint_curr - p_prev[i]
        if difference > maxdifference or difference * -1 > maxdifference:
          allGood = False
        end
        i = i + 1
      end

      if not allGood:
        struct2 = floor_corner_lift_column_extend_right(struct2)
      end

      # check whether the path involves weird turns or joint limits. final position (end of leg 3)
      joints_raa4 = [-0.8909156958209437, -1.3431089532426377, 2.273750130330221, 0.7266384798237304, 1.5611975193023682, 1.8127720355987549]
      joints_p_3 = get_inverse_kin(struct2[6], joints_raa4) # struct2[6] is p_3
      joints_p_4 = get_inverse_kin(struct2[7], joints_p_3) # struct2[7] is p_4
      joints_p_5 = get_inverse_kin(struct2[8], joints_p_4) # struct2[8] is p_5
      joints_1 = joints_p_5
      p_prev = joints_p_4
      allGood = True
      i = 0
      structlength = 6
      while i < structlength:
        joint_curr = joints_1[i]
        # check for anything that exceeds joint limits
        degreesmax = 360 * pi / 180
        if joint_curr > degreesmax or joint_curr < degreesmax * -1:
          allGood = False
        end
        # check for anything that is significantly different than the aligned approach. could indicate a twist is needed. we dont want that
        maxdifference = 150 * pi / 180
        difference = joint_curr - p_prev[i]
        if difference > maxdifference or difference * -1 > maxdifference:
          allGood = False
        end
        i = i + 1
      end

      if not allGood:
        struct2 = floor_corner_right_p_3_reduce(struct2)
      end

      # return struct2 back
      return struct2
    end

    def floor_corner_lift_column_extend_right(struct2):
      # we know that p1 cannot be accessed without a twist
      # calculate the height needed to get to p1
      liftcolumnincrement = 2.0 # mm
      enoughHeightAdded = False
      liftColumnHeightTest = 0
      while not enoughHeightAdded:
        liftColumnHeightTest = liftColumnHeightTest + liftcolumnincrement
        # set the orig_joints for p1. p1 demo was joint angles of [-0.45, -31.79, 56.47, 333.06, -130.98, 87.87] (degrees)
        # which equals [-0.007853981633974475, -0.5548401692089968, 0.985587428601197, 5.812993606692308, -2.28603225426217, 1.5336208137274159]
        orig_joints = [-0.007853981633974475, -0.5548401692089968, 0.985587428601197, 5.812993606692308, -2.28603225426217, 1.5336208137274159]
        # get the modified point:
        origp1 = struct2[0]
        testp1 = p[origp1[0], origp1[1], origp1[2] - liftColumnHeightTest / 1000.0, origp1[3], origp1[4], origp1[5]]
        testpa1 = p[origp1[0]+0.05, origp1[1]+0.05, origp1[2] - liftColumnHeightTest / 1000, origp1[3], origp1[4], origp1[5]]
        enoughHeightAdded = can_pose_be_reached_without_twist(testp1, orig_joints) and can_pose_be_reached_without_twist(testpa1, orig_joints)
      end

      origp2 = struct2[1]
      testp2 = p[origp2[0], origp2[1], origp2[2] - liftColumnHeightTest / 1000.0, origp2[3], origp2[4], origp2[5]]
      origp4 = struct2[2]
      testp4 = p[origp4[0], origp4[1], origp4[2] - liftColumnHeightTest / 1000, origp4[3], origp4[4], origp4[5]]
      origp5 = struct2[3]
      testp5 = p[origp5[0], origp5[1], origp5[2] - liftColumnHeightTest / 1000, origp5[3], origp5[4], origp5[5]]



      liftcolumnzneeded = liftColumnHeightTest
      ret = struct(point1=testp1,point2=testp2,point4=testp4,point5=testp5,point_1=struct2[4],point_2=struct2[5],point_3=struct2[6],point_4=struct2[7],point_5=struct2[8])
      return ret

    end

    # this function gets called if you are doing a left floor corner extended, and the top is too high to reach (twists, etc.)
    # this function takes the struct2 of weld points and modifies them (by subtracting from z) until the first weld point is reachable.
    # it determines the height that the lift column needs to raise to make the first point reachable
    # it then checks whether that height will allow the other points to be reachable
    # if its all good, it sets the global variable liftcolumnzneeded, modifies struct2's points, and returns struct2
    # if its not all good, then it displays an error message popup.
    def floor_corner_lift_column_extend_left(struct2):
      # we know that p1 cannot be accessed without a twist
      # calculate the height needed to get to p1
      liftcolumnincrement = 2 # mm
      enoughHeightAdded = False
      liftColumnHeightTest = 0
      while not enoughHeightAdded:
        liftColumnHeightTest = liftColumnHeightTest + liftcolumnincrement
        # set the orig_joints for p1. p1 demo was joint angles of [-0.45, -31.79, 56.47, 333.06, -130.98, 87.87] (degrees)
        # which equals [-0.007853981633974475, -0.5548401692089968, 0.985587428601197, 5.812993606692308, -2.28603225426217, 1.5336208137274159]
        orig_joints = [-0.007853981633974475, -0.5548401692089968, 0.985587428601197, 5.812993606692308, -2.28603225426217, 1.5336208137274159]
        # get the modified point:
        origp1 = struct2[0]
        testp1 = p[origp1[0], origp1[1], origp1[2] - liftColumnHeightTest / 1000, origp1[3], origp1[4], origp1[5]]
        enoughHeightAdded = can_pose_be_reached_without_twist(testp1, orig_joints)
      end


      # check whether the other 3 points are valid
      valid = True
      # get the modified point
      origp2 = struct2[1]
      testp2 = p[origp2[0], origp2[1], origp2[2] - liftColumnHeightTest / 1000, origp2[3], origp2[4], origp2[5]]
      # p2 demo was joint angles of [-0.45, -21.2, 56.98, 321.95, -130.97, 87.85] (degrees)
      # which equals [-0.007853981633974475, -0.3700098014227975, 0.9944886077863679, 5.619087526795738, -2.285857721336971, 1.5332717478770168]
      orig_joints = [-0.007853981633974475, -0.3700098014227975, 0.9944886077863679, 5.619087526795738, -2.285857721336971, 1.5332717478770168]
      valid = valid and can_pose_be_reached_without_twist(testp2, orig_joints)
      # get the modified point
      origp4 = struct2[2]
      testp4 = p[origp4[0], origp4[1], origp4[2] - liftColumnHeightTest / 1000, origp4[3], origp4[4], origp4[5]]
      # p4 demo was joint angles of [-8.62, -43.23, 99.53, 213.86, -89.19, 40.78] (degrees)
      # which equals [-0.15044738152191103, -0.7545058356371478, 1.7371262045099545, 3.7325611383150696, -1.556659159853741, 0.7117452689632868]
      orig_joints = [-0.15044738152191103, -0.7545058356371478, 1.7371262045099545, 3.7325611383150696, -1.556659159853741, 0.7117452689632868]
      valid = valid and can_pose_be_reached_without_twist(testp4, orig_joints)
      # get the modified point
      origp5 = struct2[3]
      testp5 = p[origp5[0], origp5[1], origp5[2] - liftColumnHeightTest / 1000, origp5[3], origp5[4], origp5[5]]
      # p5 demo was joint angles of [-0.59, -34.36, 77.71, 226.7, -89.18, 48.81] (degrees)
      # which equals [-0.010297442586766533, -0.5996951309852511, 1.356295361724792, 3.9566614142711405, -1.5564846269285415, 0.8518952078984314]
      orig_joints = [-0.010297442586766533, -0.5996951309852511, 1.356295361724792, 3.9566614142711405, -1.5564846269285415, 0.8518952078984314]
      valid = valid and can_pose_be_reached_without_twist(testp5, orig_joints)

      if not valid:
        # display
        popuptext = "Top of Weld is too high above robot. Cannot reach some necessary positions. Stop Program and try again with a lower top point. "
        # infinite loop
        while 1==1:
          popup(popuptext, title="Robot Positioning Warning",blocking=True)
        end
      else:
        liftcolumnzneeded = liftColumnHeightTest
        ret = struct(point1=testp1,point2=testp2,point4=testp4,point5=testp5,point_1=struct2[4],point_2=struct2[5],point_3=struct2[6],point_4=struct2[7],point_5=struct2[8])
        return ret
      end
    end

    # this function calculates whether a given pose can be reached, and if it can, whether it requires a wrist twist (from the seed joint angles)
    # arguments are target pose (p[x,y,z,rx,ry,rz]) and orig_joints which is the 6 joint angles of a pose that is close by the target pose and has the desired joint angles
    # returns true if the pose is valid and requires no twist. If pose is valid but requires a twist, returns false. If pose is invalid, returns false.
    def can_pose_be_reached_without_twist(pose, orig_joints):
      # first, determine if the pose is valid
      valid = get_inverse_kin_has_solution(pose)
      if not valid:
        return False
      end
      valid = get_inverse_kin_has_solution(pose, orig_joints)
      if not valid:
        return False
      else:
        joints_1 = get_inverse_kin(pose, orig_joints)
        #iterate through the 6 joints
        allGood = True
        i = 0
        structlength = 6
        while i < structlength:
          joint_curr = joints_1[i]
          # check for anything that exceeds joint limits
          degreesmax = 360 * pi / 180
          if joint_curr > degreesmax or joint_curr < degreesmax * -1:
            allGood = False
          end
          # check for anything that is significantly different than the aligned approach. could indicate a twist is needed. we dont want that
          maxdifference = 150 * pi / 180
          difference = joint_curr - orig_joints[i]
          if difference > maxdifference or difference * -1 > maxdifference:
            allGood = False
          end
          i = i + 1
        end
        return allGood
      end

    end

    def floor_corner_right_p_3_reduce(struct2, orig_joints):
      # we know that p_5 cannot be accessed without a twist
      # calculate the distance p_5 needs to be changed (in the direction of p_4)

      #calculate unit vector from p_5 towards p_4
      point_4 = struct2[7]
      point_5 = struct2[8]
      vecx = point_4[0] - point_5[0]
      vecy = point_4[1] - point_5[1]
      vecz = point_4[2] - point_5[2]
      mag = sqrt(vecx*vecx + vecy*vecy + vecz*vecz)
      uvx = vecx / mag
      uvy = vecy / mag
      uvz = vecz / mag

      moveincrement = 2.0 # mm
      enoughMoveAdded = False
      movement = 0

      while not enoughMoveAdded:
        movement = movement + moveincrement
        # set the orig_joints for p_4. p1 was calculated and passed into this function
        # get the modified point:
        testp_5 = p[point_5[0] + uvx*movement, point_5[1] + uvy*movement, point_5[2] + uvz*movement, point_5[3], point_5[4], point_5[5]]
        enoughMoveAdded = can_pose_be_reached_without_twist(testp_5, orig_joints)
      end

      ret = struct(point1=struct2[0],point2=struct2[1],point4=struct2[2],point5=struct2[3],point_1=struct2[4],point_2=struct2[5],point_3=struct2[6],point_4=struct2[7],point_5=testp_5)
      return ret
    end

    # this function sends a signal to turn extrusion on
    def turn_extrusion_on():
      # flush the channel
      resp0 = send_serial_signal(["u", "r", "?"])
      # send the signal
      resp1 = send_serial_signal(["u", "R", "1"])
      # if resp <> "uR1"
      if resp1 != [252,82,49]:
        # turn off extrusion and heating. inform calvin
        resp2 = send_serial_signal(["u", "R", "0"])
        resp3 = send_serial_signal(["u", "H", "0"])
        popuptext = "Error code encountered while trying to start extrusion. Find Calvin. "
        while 1==1:
          popup(popuptext, title="Extrusion Error Code",blocking=True)
          popup(resp1, blocking=True)
        end
      end
    end

    # this function sends a signal and receives a response
    # signal is a list of 3 strings, 1 character each. first is u. second is the next character. third is final character
    def send_serial_signal(signal):
      signal2char = signal[1]
      signal3char = signal[2]
      listsignal = [252, get_corr_number(signal2char), get_corr_number(signal3char)]
      resp1 = WTSerialBridge.send_command("/dev/ttyUSB0",1200, 8, "None", "One", "None", 1000, "None", "None", listsignal, True)
      return resp1
    end

    # this function converts a letter into its ascii number
    def get_corr_number(letter):
      if letter == "A":
        return 65
      elif letter == "H":
        return 72
      elif letter == "R":
        return 82
      elif letter == "M":
        return 77
      elif letter == "E":
        return 69
      elif letter == "a":
        return 97
      elif letter == "b":
        return 98
      elif letter == "h":
        return 104
      elif letter == "r":
        return 114
      elif letter == "s":
        return 115
      elif letter == "m":
        return 109
      elif letter == "0":
        return 48
      elif letter == "1":
        return 49
      elif letter == "2":
        return 50
      elif letter == "3":
        return 51
      elif letter == "4":
        return 52
      elif letter == "5":
        return 53
      elif letter == "6":
        return 54
      elif letter == "7":
        return 55
      elif letter == "8":
        return 56
      elif letter == "9":
        return 57
      elif letter == "?":
        return 63
      end
    end

